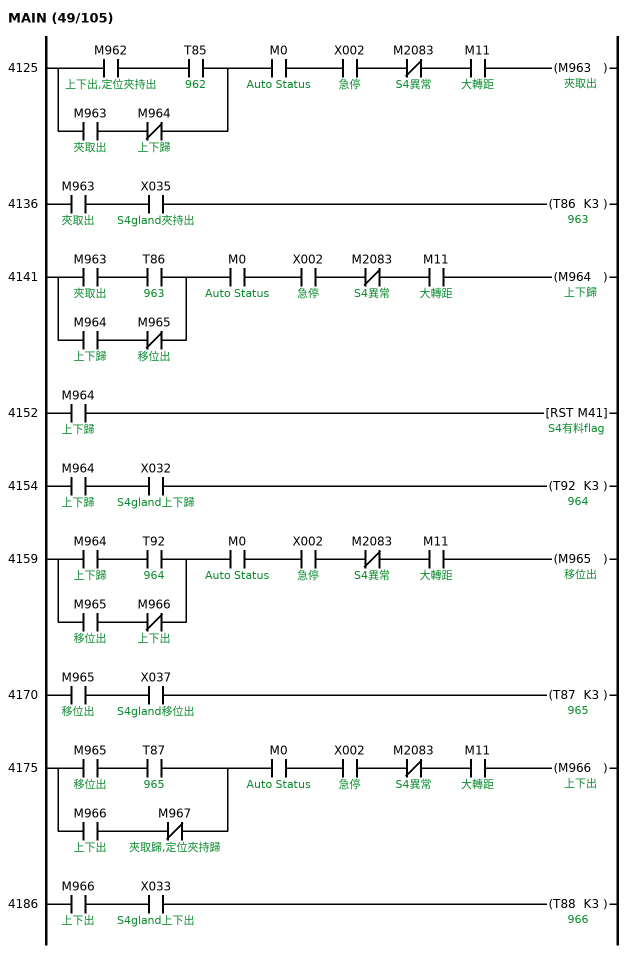
[picture p48: ladder of MAIN, rungs at steps 4125 to 4186]
4125  LD      M962  ; 上下出,定位夾持出
      AND     T85  ; 962
      LD      M963  ; 夾取出
      ANI     M964  ; 上下歸
      ORB
      AND     M0  ; Auto Status
      AND     X002  ; 急停
      ANI     M2083  ; S4異常
      AND     M11  ; 大轉距
      OUT     M963  ; 夾取出
4136  LD      M963  ; 夾取出
      AND     X035  ; S4gland夾持出
      OUT     T86 K3  ; 963
4141  LD      M963  ; 夾取出
      AND     T86  ; 963
      LD      M964  ; 上下歸
      ANI     M965  ; 移位出
      ORB
      AND     M0  ; Auto Status
      AND     X002  ; 急停
      ANI     M2083  ; S4異常
      AND     M11  ; 大轉距
      OUT     M964  ; 上下歸
4152  LD      M964  ; 上下歸
      RST     M41  ; S4有料flag
4154  LD      M964  ; 上下歸
      AND     X032  ; S4gland上下歸
      OUT     T92 K3  ; 964
4159  LD      M964  ; 上下歸
      AND     T92  ; 964
      LD      M965  ; 移位出
      ANI     M966  ; 上下出
      ORB
      AND     M0  ; Auto Status
      AND     X002  ; 急停
      ANI     M2083  ; S4異常
      AND     M11  ; 大轉距
      OUT     M965  ; 移位出
4170  LD      M965  ; 移位出
      AND     X037  ; S4gland移位出
      OUT     T87 K3  ; 965
4175  LD      M965  ; 移位出
      AND     T87  ; 965
      LD      M966  ; 上下出
      ANI     M967  ; 夾取歸,定位夾持歸
      ORB
      AND     M0  ; Auto Status
      AND     X002  ; 急停
      ANI     M2083  ; S4異常
      AND     M11  ; 大轉距
      OUT     M966  ; 上下出
4186  LD      M966  ; 上下出
      AND     X033  ; S4gland上下出
      OUT     T88 K3  ; 966
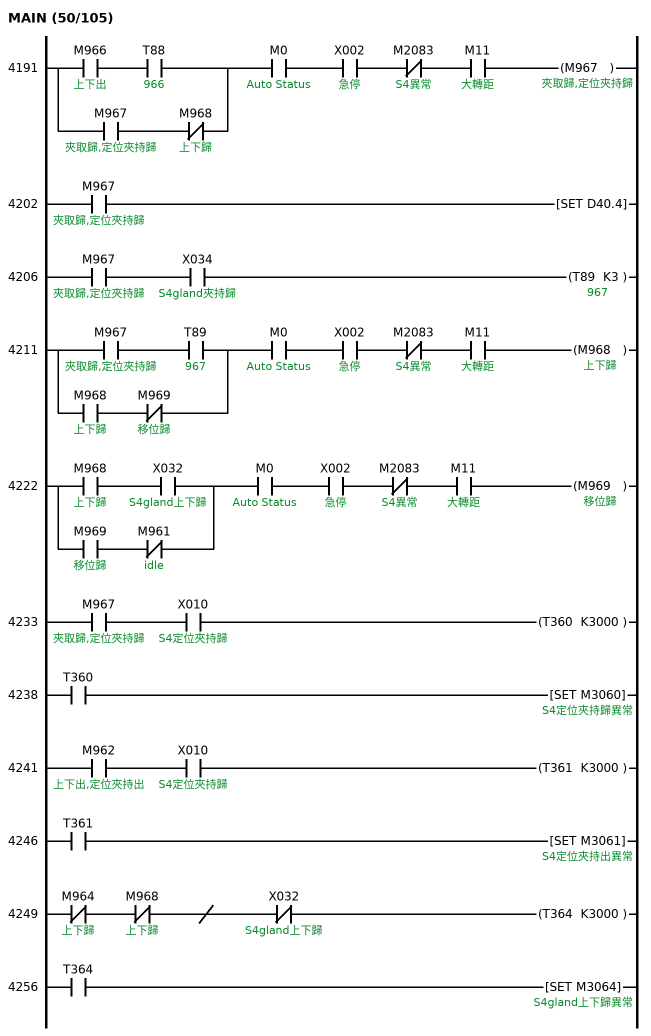
4191  LD      M966  ; 上下出
      AND     T88  ; 966
      LD      M967  ; 夾取歸,定位夾持歸
      ANI     M968  ; 上下歸
      ORB
      AND     M0  ; Auto Status
      AND     X002  ; 急停
      ANI     M2083  ; S4異常
      AND     M11  ; 大轉距
      OUT     M967  ; 夾取歸,定位夾持歸
4202  LD      M967  ; 夾取歸,定位夾持歸
      SET     D40.4
4206  LD      M967  ; 夾取歸,定位夾持歸
      AND     X034  ; S4gland夾持歸
      OUT     T89 K3  ; 967
4211  LD      M967  ; 夾取歸,定位夾持歸
      AND     T89  ; 967
      LD      M968  ; 上下歸
      ANI     M969  ; 移位歸
      ORB
      AND     M0  ; Auto Status
      AND     X002  ; 急停
      ANI     M2083  ; S4異常
      AND     M11  ; 大轉距
      OUT     M968  ; 上下歸
4222  LD      M968  ; 上下歸
      AND     X032  ; S4gland上下歸
      LD      M969  ; 移位歸
      ANI     M961  ; idle
      ORB
      AND     M0  ; Auto Status
      AND     X002  ; 急停
      ANI     M2083  ; S4異常
      AND     M11  ; 大轉距
      OUT     M969  ; 移位歸
4233  LD      M967  ; 夾取歸,定位夾持歸
      AND     X010  ; S4定位夾持歸
      OUT     T360 K3000
4238  LD      T360
      SET     M3060  ; S4定位夾持歸異常
4241  LD      M962  ; 上下出,定位夾持出
      AND     X010  ; S4定位夾持歸
      OUT     T361 K3000
4246  LD      T361
      SET     M3061  ; S4定位夾持出異常
4249  LDI     M964  ; 上下歸
      ANI     M968  ; 上下歸
      INV
      ANI     X032  ; S4gland上下歸
      OUT     T364 K3000
4256  LD      T364
      SET     M3064  ; S4gland上下歸異常
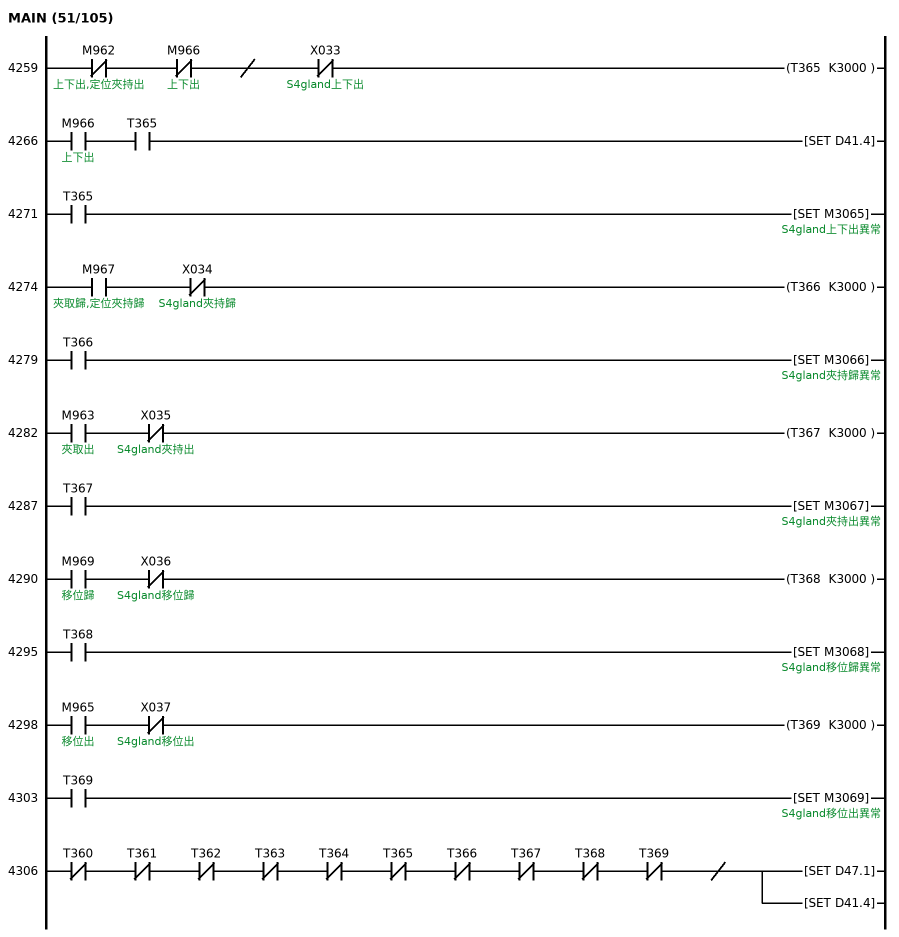
4259  LDI     M962  ; 上下出,定位夾持出
      ANI     M966  ; 上下出
      INV
      ANI     X033  ; S4gland上下出
      OUT     T365 K3000
4266  LD      M966  ; 上下出
      AND     T365
      SET     D41.4
4271  LD      T365
      SET     M3065  ; S4gland上下出異常
4274  LD      M967  ; 夾取歸,定位夾持歸
      ANI     X034  ; S4gland夾持歸
      OUT     T366 K3000
4279  LD      T366
      SET     M3066  ; S4gland夾持歸異常
4282  LD      M963  ; 夾取出
      ANI     X035  ; S4gland夾持出
      OUT     T367 K3000
4287  LD      T367
      SET     M3067  ; S4gland夾持出異常
4290  LD      M969  ; 移位歸
      ANI     X036  ; S4gland移位歸
      OUT     T368 K3000
4295  LD      T368
      SET     M3068  ; S4gland移位歸異常
4298  LD      M965  ; 移位出
      ANI     X037  ; S4gland移位出
      OUT     T369 K3000
4303  LD      T369
      SET     M3069  ; S4gland移位出異常
4306  LDI     T360
      ANI     T361
      ANI     T362
      ANI     T363
      ANI     T364
      ANI     T365
      ANI     T366
      ANI     T367
      ANI     T368
      ANI     T369
      INV
      SET     D47.1
      SET     D41.4
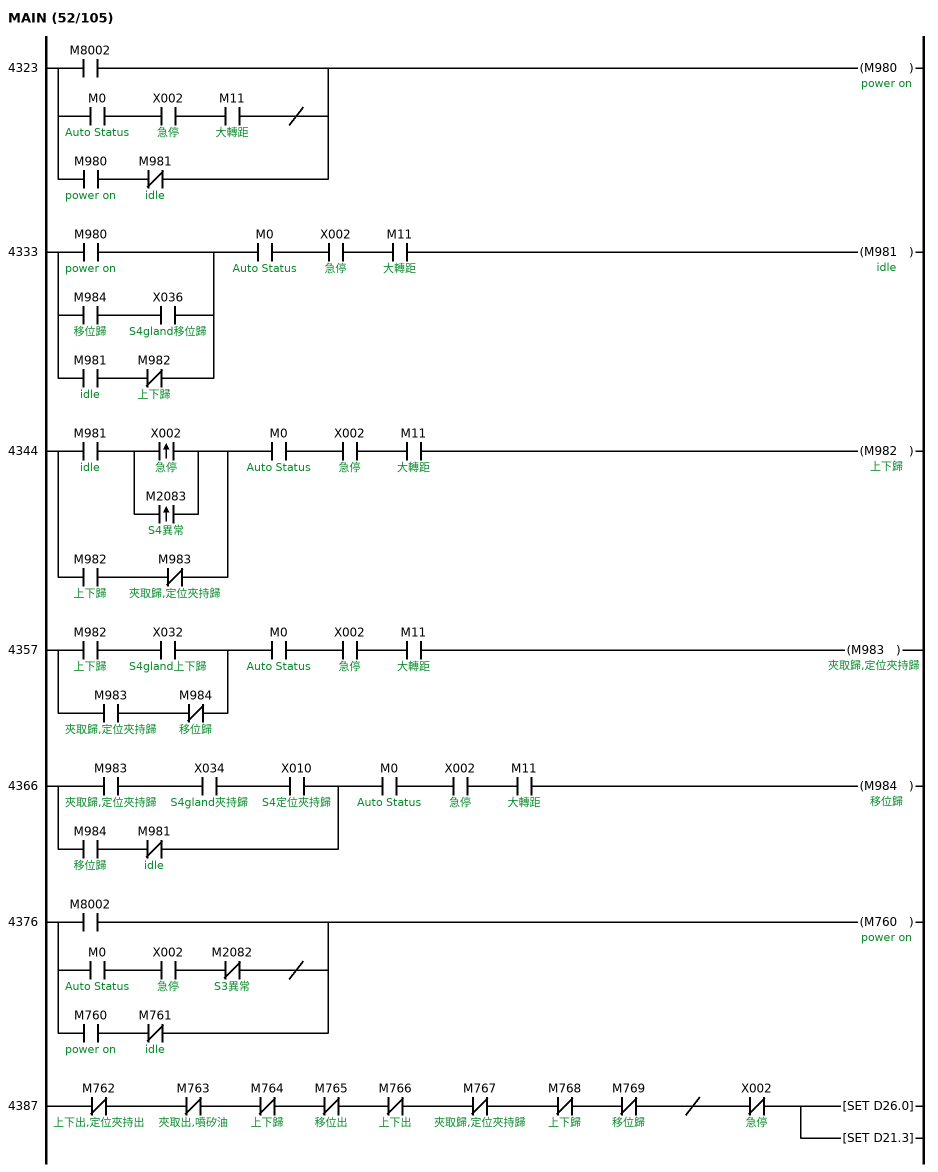
4323  LD      M8002
      LD      M0  ; Auto Status
      AND     X002  ; 急停
      AND     M11  ; 大轉距
      INV
      ORB
      LD      M980  ; power on
      ANI     M981  ; idle
      ORB
      OUT     M980  ; power on
4333  LD      M980  ; power on
      LD      M984  ; 移位歸
      AND     X036  ; S4gland移位歸
      ORB
      LD      M981  ; idle
      ANI     M982  ; 上下歸
      ORB
      AND     M0  ; Auto Status
      AND     X002  ; 急停
      AND     M11  ; 大轉距
      OUT     M981  ; idle
4344  LD      M981  ; idle
      LDP     X002  ; 急停
      ORP     M2083  ; S4異常
      ANB
      LD      M982  ; 上下歸
      ANI     M983  ; 夾取歸,定位夾持歸
      ORB
      AND     M0  ; Auto Status
      AND     X002  ; 急停
      AND     M11  ; 大轉距
      OUT     M982  ; 上下歸
4357  LD      M982  ; 上下歸
      AND     X032  ; S4gland上下歸
      LD      M983  ; 夾取歸,定位夾持歸
      ANI     M984  ; 移位歸
      ORB
      AND     M0  ; Auto Status
      AND     X002  ; 急停
      AND     M11  ; 大轉距
      OUT     M983  ; 夾取歸,定位夾持歸
4366  LD      M983  ; 夾取歸,定位夾持歸
      AND     X034  ; S4gland夾持歸
      AND     X010  ; S4定位夾持歸
      LD      M984  ; 移位歸
      ANI     M981  ; idle
      ORB
      AND     M0  ; Auto Status
      AND     X002  ; 急停
      AND     M11  ; 大轉距
      OUT     M984  ; 移位歸
4376  LD      M8002
      LD      M0  ; Auto Status
      AND     X002  ; 急停
      ANI     M2082  ; S3異常
      INV
      ORB
      LD      M760  ; power on
      ANI     M761  ; idle
      ORB
      OUT     M760  ; power on
4387  LDI     M762  ; 上下出,定位夾持出
      ANI     M763  ; 夾取出,噴矽油
      ANI     M764  ; 上下歸
      ANI     M765  ; 移位出
      ANI     M766  ; 上下出
      ANI     M767  ; 夾取歸,定位夾持歸
      ANI     M768  ; 上下歸
      ANI     M769  ; 移位歸
      INV
      ANI     X002  ; 急停
      SET     D26.0
      SET     D21.3
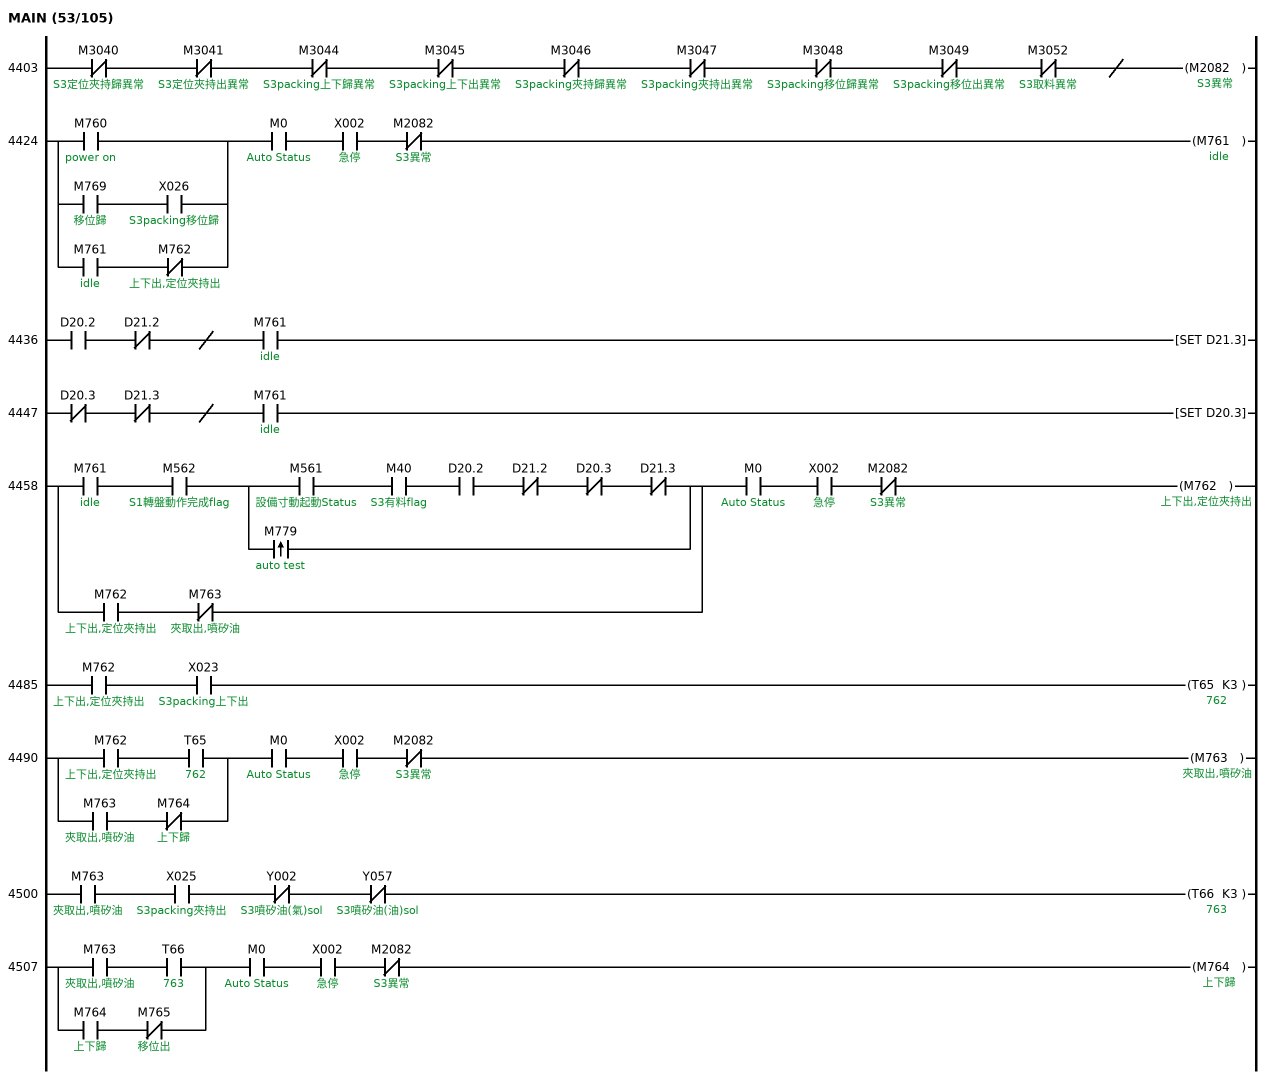
4403  LDI     M3040  ; S3定位夾持歸異常
      ANI     M3041  ; S3定位夾持出異常
      ANI     M3044  ; S3packing上下歸異常
      ANI     M3045  ; S3packing上下出異常
      ANI     M3046  ; S3packing夾持歸異常
      ANI     M3047  ; S3packing夾持出異常
      ANI     M3048  ; S3packing移位歸異常
      ANI     M3049  ; S3packing移位出異常
      ANI     M3052  ; S3取料異常
      INV
      OUT     M2082  ; S3異常
4424  LD      M760  ; power on
      LD      M769  ; 移位歸
      AND     X026  ; S3packing移位歸
      ORB
      LD      M761  ; idle
      ANI     M762  ; 上下出,定位夾持出
      ORB
      AND     M0  ; Auto Status
      AND     X002  ; 急停
      ANI     M2082  ; S3異常
      OUT     M761  ; idle
4436  LD      D20.2
      ANI     D21.2
      INV
      AND     M761  ; idle
      SET     D21.3
4447  LDI     D20.3
      ANI     D21.3
      INV
      AND     M761  ; idle
      SET     D20.3
4458  LD      M761  ; idle
      AND     M562  ; S1轉盤動作完成flag
      LD      M561  ; 設備寸動起動Status
      AND     M40  ; S3有料flag
      AND     D20.2
      ANI     D21.2
      ANI     D20.3
      ANI     D21.3
      ORP     M779  ; auto test
      ANB
      LD      M762  ; 上下出,定位夾持出
      ANI     M763  ; 夾取出,噴矽油
      ORB
      AND     M0  ; Auto Status
      AND     X002  ; 急停
      ANI     M2082  ; S3異常
      OUT     M762  ; 上下出,定位夾持出
4485  LD      M762  ; 上下出,定位夾持出
      AND     X023  ; S3packing上下出
      OUT     T65 K3  ; 762
4490  LD      M762  ; 上下出,定位夾持出
      AND     T65  ; 762
      LD      M763  ; 夾取出,噴矽油
      ANI     M764  ; 上下歸
      ORB
      AND     M0  ; Auto Status
      AND     X002  ; 急停
      ANI     M2082  ; S3異常
      OUT     M763  ; 夾取出,噴矽油
4500  LD      M763  ; 夾取出,噴矽油
      AND     X025  ; S3packing夾持出
      ANI     Y002  ; S3噴矽油(氣)sol
      ANI     Y057  ; S3噴矽油(油)sol
      OUT     T66 K3  ; 763
4507  LD      M763  ; 夾取出,噴矽油
      AND     T66  ; 763
      LD      M764  ; 上下歸
      ANI     M765  ; 移位出
      ORB
      AND     M0  ; Auto Status
      AND     X002  ; 急停
      ANI     M2082  ; S3異常
      OUT     M764  ; 上下歸
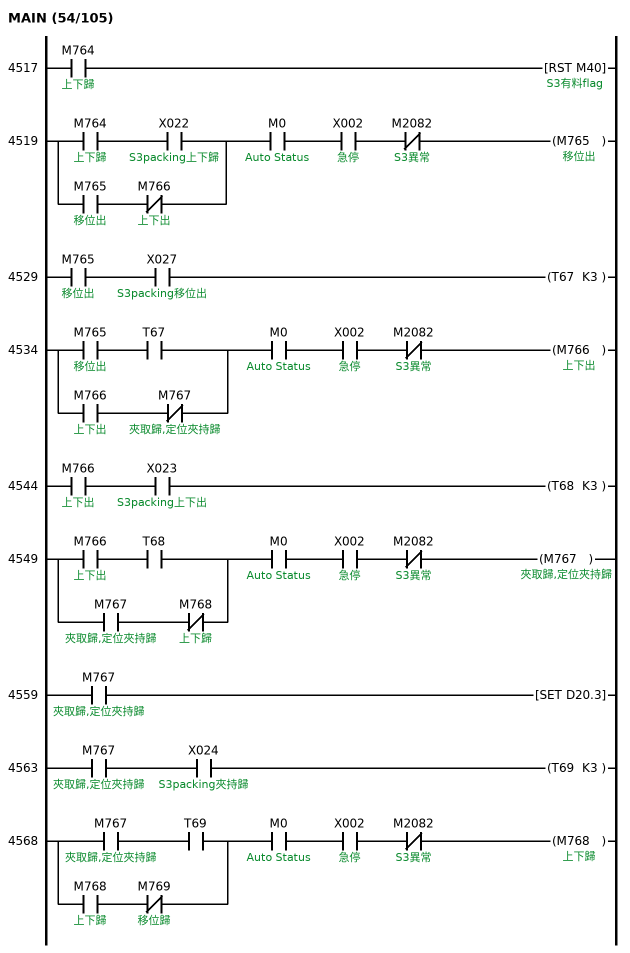
4517  LD      M764  ; 上下歸
      RST     M40  ; S3有料flag
4519  LD      M764  ; 上下歸
      AND     X022  ; S3packing上下歸
      LD      M765  ; 移位出
      ANI     M766  ; 上下出
      ORB
      AND     M0  ; Auto Status
      AND     X002  ; 急停
      ANI     M2082  ; S3異常
      OUT     M765  ; 移位出
4529  LD      M765  ; 移位出
      AND     X027  ; S3packing移位出
      OUT     T67 K3
4534  LD      M765  ; 移位出
      AND     T67
      LD      M766  ; 上下出
      ANI     M767  ; 夾取歸,定位夾持歸
      ORB
      AND     M0  ; Auto Status
      AND     X002  ; 急停
      ANI     M2082  ; S3異常
      OUT     M766  ; 上下出
4544  LD      M766  ; 上下出
      AND     X023  ; S3packing上下出
      OUT     T68 K3
4549  LD      M766  ; 上下出
      AND     T68
      LD      M767  ; 夾取歸,定位夾持歸
      ANI     M768  ; 上下歸
      ORB
      AND     M0  ; Auto Status
      AND     X002  ; 急停
      ANI     M2082  ; S3異常
      OUT     M767  ; 夾取歸,定位夾持歸
4559  LD      M767  ; 夾取歸,定位夾持歸
      SET     D20.3
4563  LD      M767  ; 夾取歸,定位夾持歸
      AND     X024  ; S3packing夾持歸
      OUT     T69 K3
4568  LD      M767  ; 夾取歸,定位夾持歸
      AND     T69
      LD      M768  ; 上下歸
      ANI     M769  ; 移位歸
      ORB
      AND     M0  ; Auto Status
      AND     X002  ; 急停
      ANI     M2082  ; S3異常
      OUT     M768  ; 上下歸
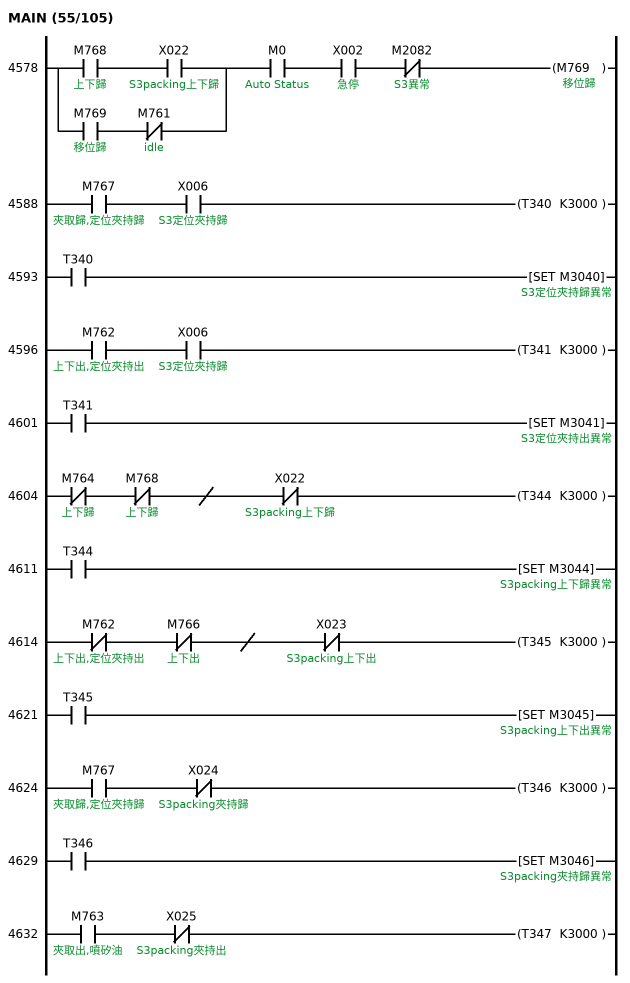
4578  LD      M768  ; 上下歸
      AND     X022  ; S3packing上下歸
      LD      M769  ; 移位歸
      ANI     M761  ; idle
      ORB
      AND     M0  ; Auto Status
      AND     X002  ; 急停
      ANI     M2082  ; S3異常
      OUT     M769  ; 移位歸
4588  LD      M767  ; 夾取歸,定位夾持歸
      AND     X006  ; S3定位夾持歸
      OUT     T340 K3000
4593  LD      T340
      SET     M3040  ; S3定位夾持歸異常
4596  LD      M762  ; 上下出,定位夾持出
      AND     X006  ; S3定位夾持歸
      OUT     T341 K3000
4601  LD      T341
      SET     M3041  ; S3定位夾持出異常
4604  LDI     M764  ; 上下歸
      ANI     M768  ; 上下歸
      INV
      ANI     X022  ; S3packing上下歸
      OUT     T344 K3000
4611  LD      T344
      SET     M3044  ; S3packing上下歸異常
4614  LDI     M762  ; 上下出,定位夾持出
      ANI     M766  ; 上下出
      INV
      ANI     X023  ; S3packing上下出
      OUT     T345 K3000
4621  LD      T345
      SET     M3045  ; S3packing上下出異常
4624  LD      M767  ; 夾取歸,定位夾持歸
      ANI     X024  ; S3packing夾持歸
      OUT     T346 K3000
4629  LD      T346
      SET     M3046  ; S3packing夾持歸異常
4632  LD      M763  ; 夾取出,噴矽油
      ANI     X025  ; S3packing夾持出
      OUT     T347 K3000
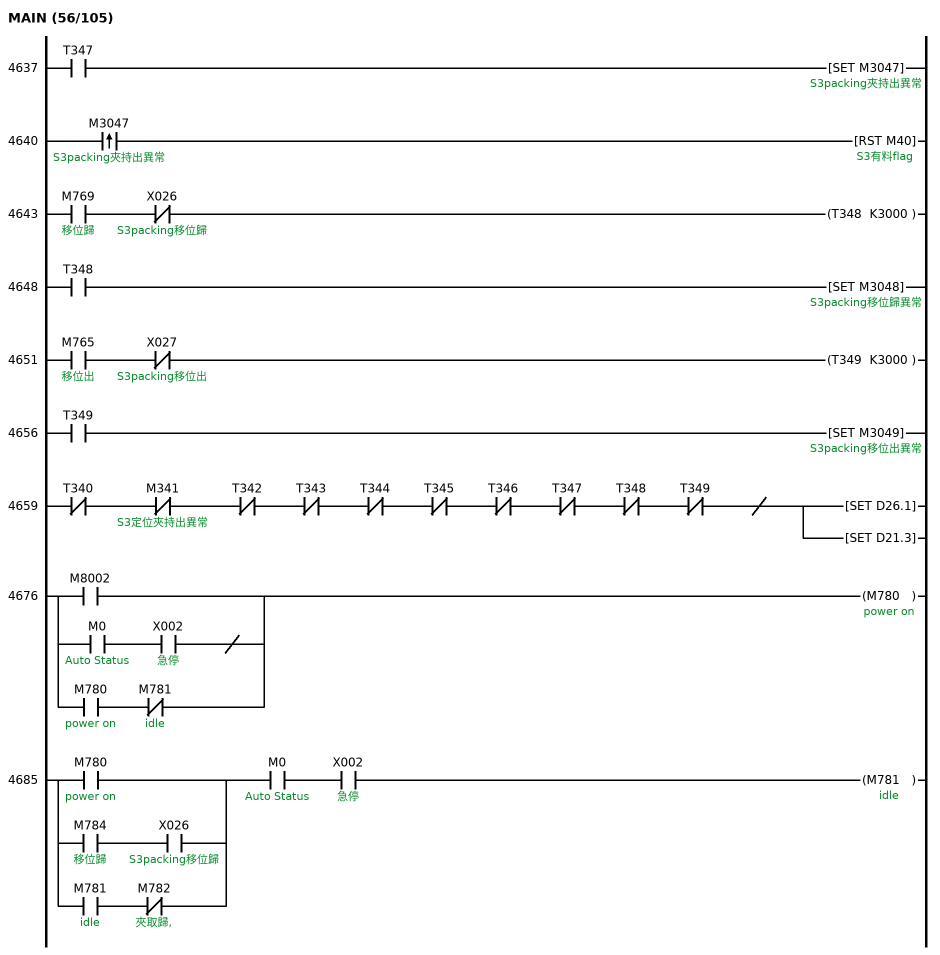
4637  LD      T347
      SET     M3047  ; S3packing夾持出異常
4640  LDP     M3047  ; S3packing夾持出異常
      RST     M40  ; S3有料flag
4643  LD      M769  ; 移位歸
      ANI     X026  ; S3packing移位歸
      OUT     T348 K3000
4648  LD      T348
      SET     M3048  ; S3packing移位歸異常
4651  LD      M765  ; 移位出
      ANI     X027  ; S3packing移位出
      OUT     T349 K3000
4656  LD      T349
      SET     M3049  ; S3packing移位出異常
4659  LDI     T340
      ANI     M341  ; S3定位夾持出異常
      ANI     T342
      ANI     T343
      ANI     T344
      ANI     T345
      ANI     T346
      ANI     T347
      ANI     T348
      ANI     T349
      INV
      SET     D26.1
      SET     D21.3
4676  LD      M8002
      LD      M0  ; Auto Status
      AND     X002  ; 急停
      INV
      ORB
      LD      M780  ; power on
      ANI     M781  ; idle
      ORB
      OUT     M780  ; power on
4685  LD      M780  ; power on
      LD      M784  ; 移位歸
      AND     X026  ; S3packing移位歸
      ORB
      LD      M781  ; idle
      ANI     M782  ; 夾取歸,
      ORB
      AND     M0  ; Auto Status
      AND     X002  ; 急停
      OUT     M781  ; idle
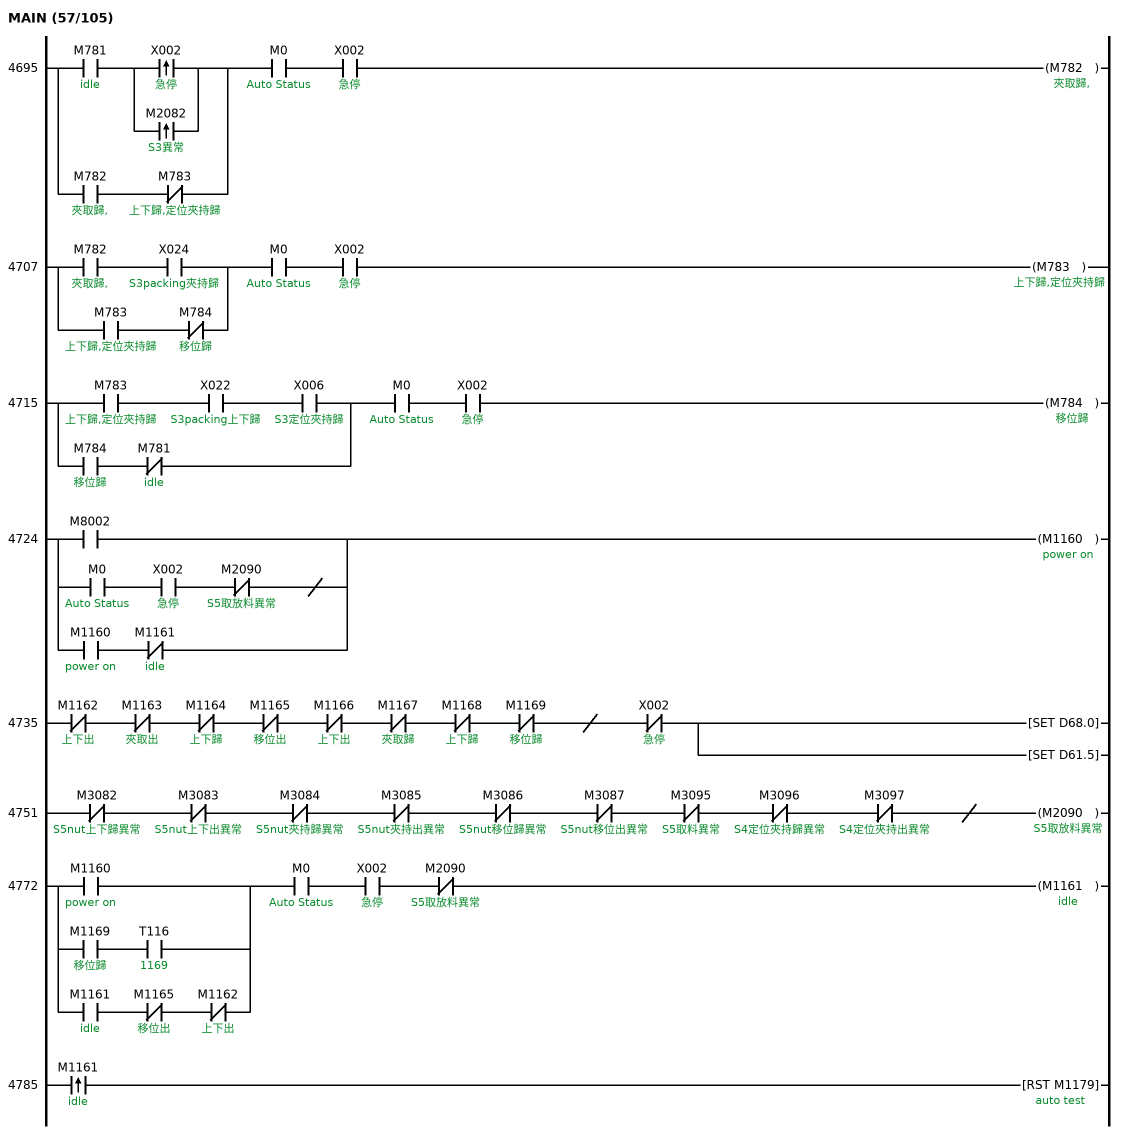
4695  LD      M781  ; idle
      LDP     X002  ; 急停
      ORP     M2082  ; S3異常
      ANB
      LD      M782  ; 夾取歸,
      ANI     M783  ; 上下歸,定位夾持歸
      ORB
      AND     M0  ; Auto Status
      AND     X002  ; 急停
      OUT     M782  ; 夾取歸,
4707  LD      M782  ; 夾取歸,
      AND     X024  ; S3packing夾持歸
      LD      M783  ; 上下歸,定位夾持歸
      ANI     M784  ; 移位歸
      ORB
      AND     M0  ; Auto Status
      AND     X002  ; 急停
      OUT     M783  ; 上下歸,定位夾持歸
4715  LD      M783  ; 上下歸,定位夾持歸
      AND     X022  ; S3packing上下歸
      AND     X006  ; S3定位夾持歸
      LD      M784  ; 移位歸
      ANI     M781  ; idle
      ORB
      AND     M0  ; Auto Status
      AND     X002  ; 急停
      OUT     M784  ; 移位歸
4724  LD      M8002
      LD      M0  ; Auto Status
      AND     X002  ; 急停
      ANI     M2090  ; S5取放料異常
      INV
      ORB
      LD      M1160  ; power on
      ANI     M1161  ; idle
      ORB
      OUT     M1160  ; power on
4735  LDI     M1162  ; 上下出
      ANI     M1163  ; 夾取出
      ANI     M1164  ; 上下歸
      ANI     M1165  ; 移位出
      ANI     M1166  ; 上下出
      ANI     M1167  ; 夾取歸
      ANI     M1168  ; 上下歸
      ANI     M1169  ; 移位歸
      INV
      ANI     X002  ; 急停
      SET     D68.0
      SET     D61.5
4751  LDI     M3082  ; S5nut上下歸異常
      ANI     M3083  ; S5nut上下出異常
      ANI     M3084  ; S5nut夾持歸異常
      ANI     M3085  ; S5nut夾持出異常
      ANI     M3086  ; S5nut移位歸異常
      ANI     M3087  ; S5nut移位出異常
      ANI     M3095  ; S5取料異常
      ANI     M3096  ; S4定位夾持歸異常
      ANI     M3097  ; S4定位夾持出異常
      INV
      OUT     M2090  ; S5取放料異常
4772  LD      M1160  ; power on
      LD      M1169  ; 移位歸
      AND     T116  ; 1169
      ORB
      LD      M1161  ; idle
      ANI     M1165  ; 移位出
      ANI     M1162  ; 上下出
      ORB
      AND     M0  ; Auto Status
      AND     X002  ; 急停
      ANI     M2090  ; S5取放料異常
      OUT     M1161  ; idle
4785  LDP     M1161  ; idle
      RST     M1179  ; auto test
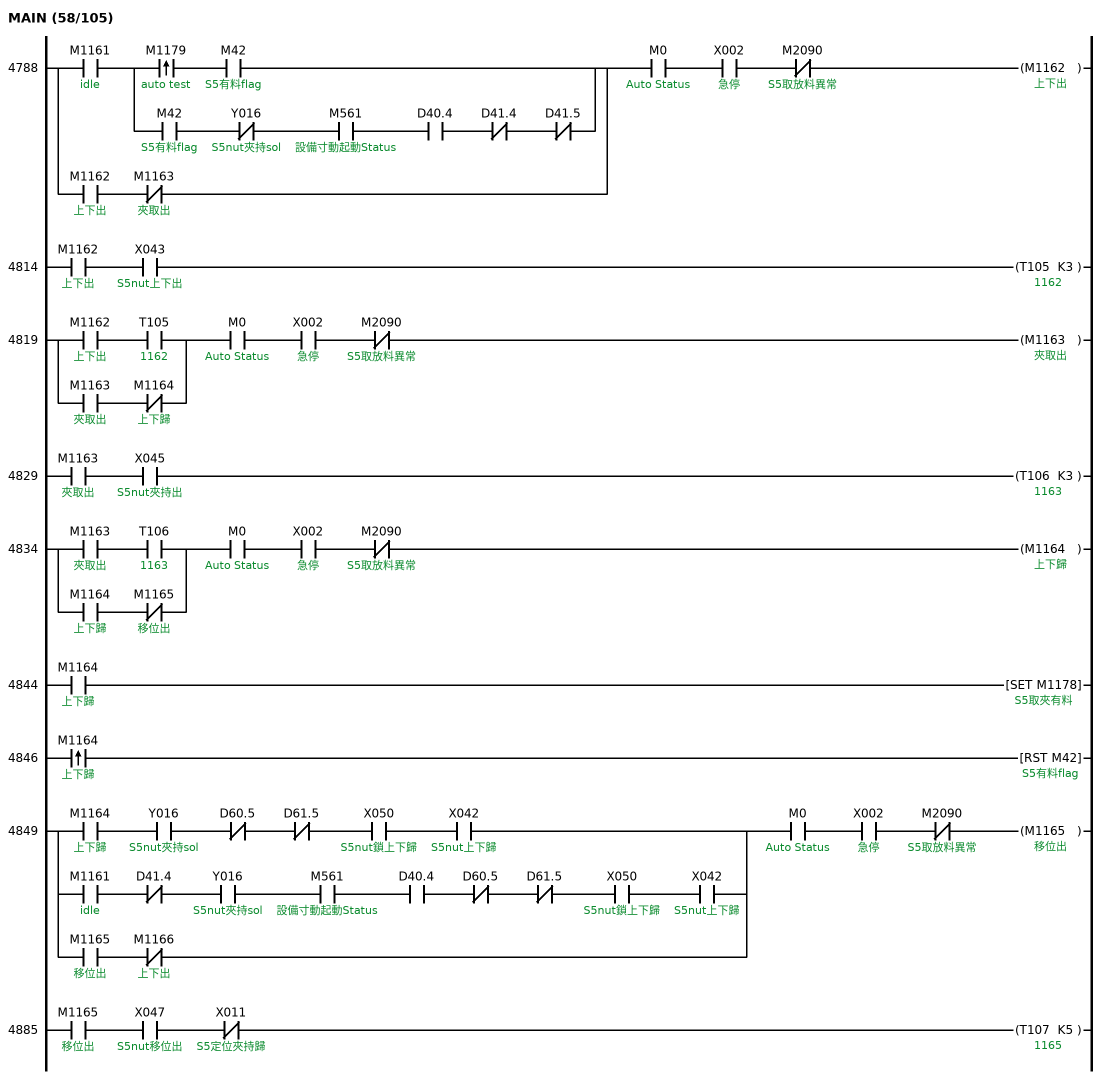
4788  LD      M1161  ; idle
      LDP     M1179  ; auto test
      AND     M42  ; S5有料flag
      LD      M42  ; S5有料flag
      ANI     Y016  ; S5nut夾持sol
      AND     M561  ; 設備寸動起動Status
      AND     D40.4
      ANI     D41.4
      ANI     D41.5
      ORB
      ANB
      LD      M1162  ; 上下出
      ANI     M1163  ; 夾取出
      ORB
      AND     M0  ; Auto Status
      AND     X002  ; 急停
      ANI     M2090  ; S5取放料異常
      OUT     M1162  ; 上下出
4814  LD      M1162  ; 上下出
      AND     X043  ; S5nut上下出
      OUT     T105 K3  ; 1162
4819  LD      M1162  ; 上下出
      AND     T105  ; 1162
      LD      M1163  ; 夾取出
      ANI     M1164  ; 上下歸
      ORB
      AND     M0  ; Auto Status
      AND     X002  ; 急停
      ANI     M2090  ; S5取放料異常
      OUT     M1163  ; 夾取出
4829  LD      M1163  ; 夾取出
      AND     X045  ; S5nut夾持出
      OUT     T106 K3  ; 1163
4834  LD      M1163  ; 夾取出
      AND     T106  ; 1163
      LD      M1164  ; 上下歸
      ANI     M1165  ; 移位出
      ORB
      AND     M0  ; Auto Status
      AND     X002  ; 急停
      ANI     M2090  ; S5取放料異常
      OUT     M1164  ; 上下歸
4844  LD      M1164  ; 上下歸
      SET     M1178  ; S5取夾有料
4846  LDP     M1164  ; 上下歸
      RST     M42  ; S5有料flag
4849  LD      M1164  ; 上下歸
      AND     Y016  ; S5nut夾持sol
      ANI     D60.5
      ANI     D61.5
      AND     X050  ; S5nut鎖上下歸
      AND     X042  ; S5nut上下歸
      LD      M1161  ; idle
      ANI     D41.4
      AND     Y016  ; S5nut夾持sol
      AND     M561  ; 設備寸動起動Status
      AND     D40.4
      ANI     D60.5
      ANI     D61.5
      AND     X050  ; S5nut鎖上下歸
      AND     X042  ; S5nut上下歸
      ORB
      LD      M1165  ; 移位出
      ANI     M1166  ; 上下出
      ORB
      AND     M0  ; Auto Status
      AND     X002  ; 急停
      ANI     M2090  ; S5取放料異常
      OUT     M1165  ; 移位出
4885  LD      M1165  ; 移位出
      AND     X047  ; S5nut移位出
      ANI     X011  ; S5定位夾持歸
      OUT     T107 K5  ; 1165
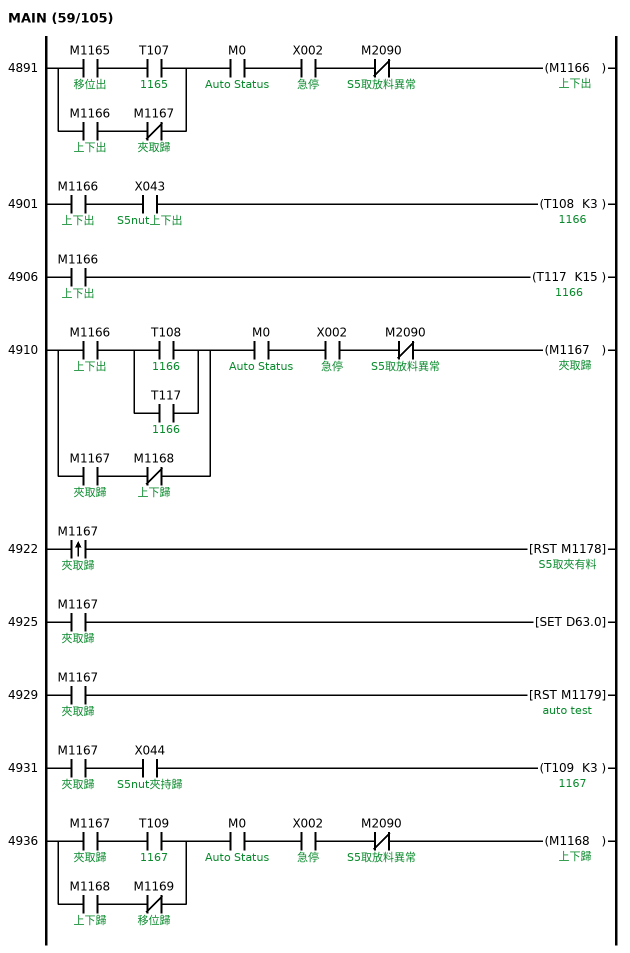
4891  LD      M1165  ; 移位出
      AND     T107  ; 1165
      LD      M1166  ; 上下出
      ANI     M1167  ; 夾取歸
      ORB
      AND     M0  ; Auto Status
      AND     X002  ; 急停
      ANI     M2090  ; S5取放料異常
      OUT     M1166  ; 上下出
4901  LD      M1166  ; 上下出
      AND     X043  ; S5nut上下出
      OUT     T108 K3  ; 1166
4906  LD      M1166  ; 上下出
      OUT     T117 K15  ; 1166
4910  LD      M1166  ; 上下出
      LD      T108  ; 1166
      OR      T117  ; 1166
      ANB
      LD      M1167  ; 夾取歸
      ANI     M1168  ; 上下歸
      ORB
      AND     M0  ; Auto Status
      AND     X002  ; 急停
      ANI     M2090  ; S5取放料異常
      OUT     M1167  ; 夾取歸
4922  LDP     M1167  ; 夾取歸
      RST     M1178  ; S5取夾有料
4925  LD      M1167  ; 夾取歸
      SET     D63.0
4929  LD      M1167  ; 夾取歸
      RST     M1179  ; auto test
4931  LD      M1167  ; 夾取歸
      AND     X044  ; S5nut夾持歸
      OUT     T109 K3  ; 1167
4936  LD      M1167  ; 夾取歸
      AND     T109  ; 1167
      LD      M1168  ; 上下歸
      ANI     M1169  ; 移位歸
      ORB
      AND     M0  ; Auto Status
      AND     X002  ; 急停
      ANI     M2090  ; S5取放料異常
      OUT     M1168  ; 上下歸
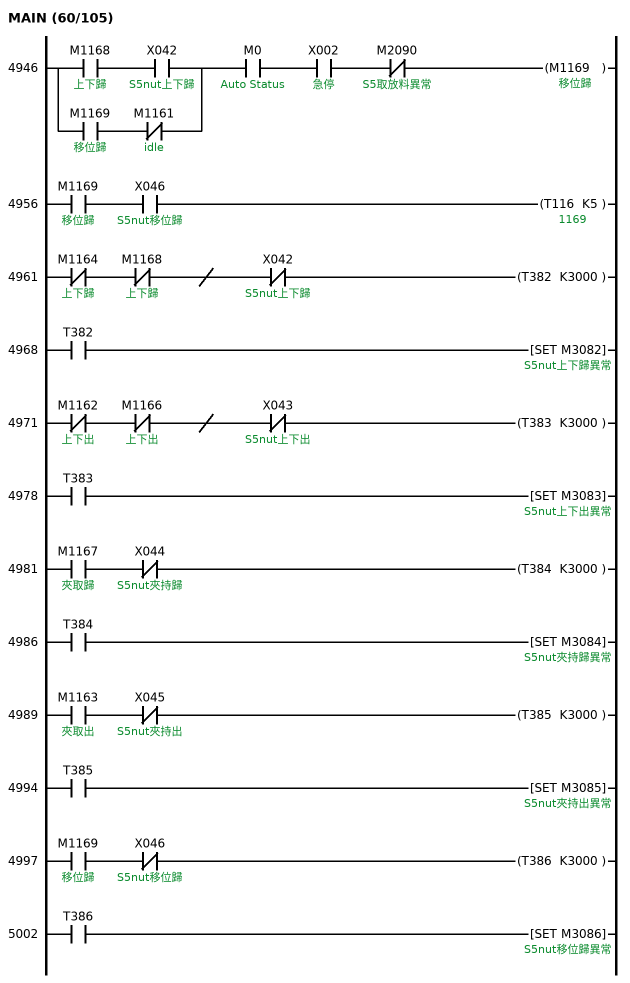
4946  LD      M1168  ; 上下歸
      AND     X042  ; S5nut上下歸
      LD      M1169  ; 移位歸
      ANI     M1161  ; idle
      ORB
      AND     M0  ; Auto Status
      AND     X002  ; 急停
      ANI     M2090  ; S5取放料異常
      OUT     M1169  ; 移位歸
4956  LD      M1169  ; 移位歸
      AND     X046  ; S5nut移位歸
      OUT     T116 K5  ; 1169
4961  LDI     M1164  ; 上下歸
      ANI     M1168  ; 上下歸
      INV
      ANI     X042  ; S5nut上下歸
      OUT     T382 K3000
4968  LD      T382
      SET     M3082  ; S5nut上下歸異常
4971  LDI     M1162  ; 上下出
      ANI     M1166  ; 上下出
      INV
      ANI     X043  ; S5nut上下出
      OUT     T383 K3000
4978  LD      T383
      SET     M3083  ; S5nut上下出異常
4981  LD      M1167  ; 夾取歸
      ANI     X044  ; S5nut夾持歸
      OUT     T384 K3000
4986  LD      T384
      SET     M3084  ; S5nut夾持歸異常
4989  LD      M1163  ; 夾取出
      ANI     X045  ; S5nut夾持出
      OUT     T385 K3000
4994  LD      T385
      SET     M3085  ; S5nut夾持出異常
4997  LD      M1169  ; 移位歸
      ANI     X046  ; S5nut移位歸
      OUT     T386 K3000
5002  LD      T386
      SET     M3086  ; S5nut移位歸異常
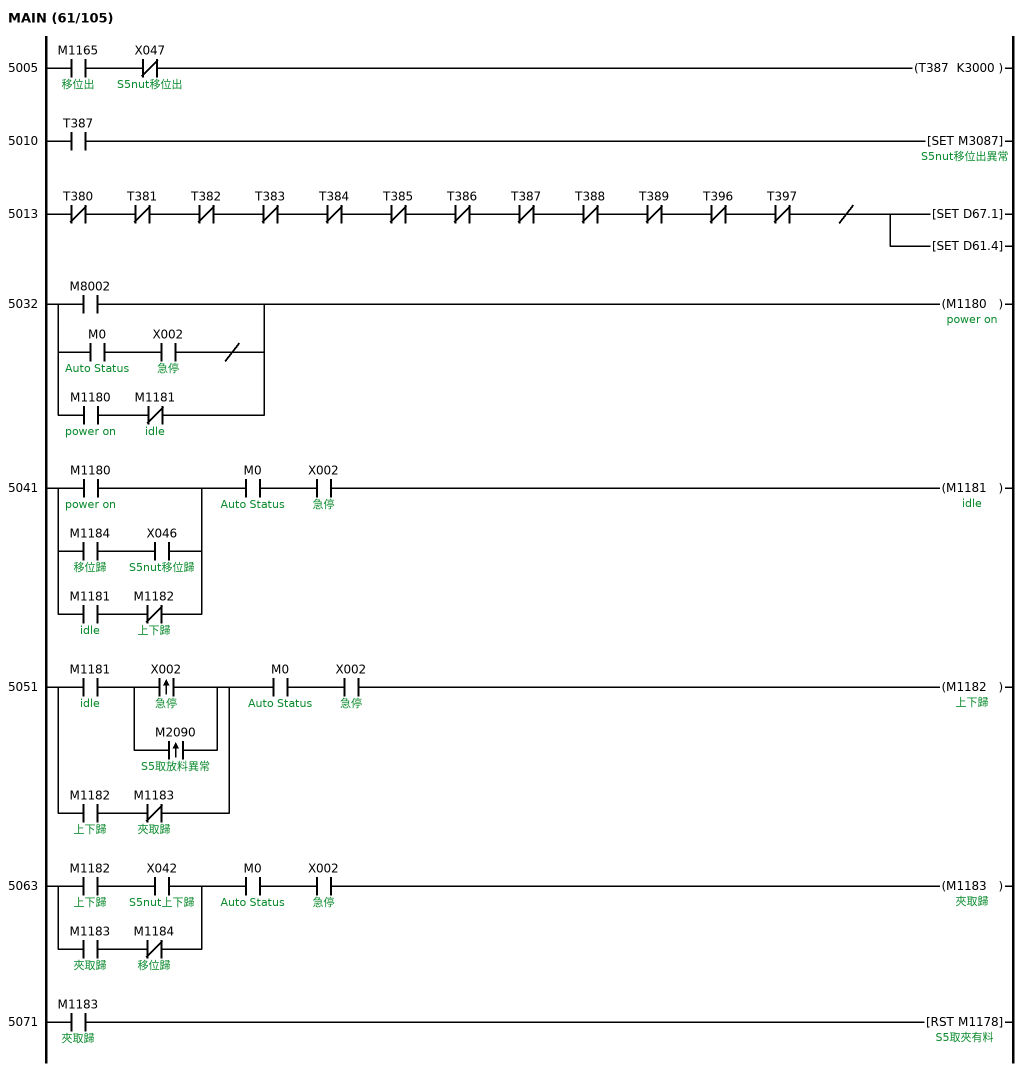
5005  LD      M1165  ; 移位出
      ANI     X047  ; S5nut移位出
      OUT     T387 K3000
5010  LD      T387
      SET     M3087  ; S5nut移位出異常
5013  LDI     T380
      ANI     T381
      ANI     T382
      ANI     T383
      ANI     T384
      ANI     T385
      ANI     T386
      ANI     T387
      ANI     T388
      ANI     T389
      ANI     T396
      ANI     T397
      INV
      SET     D67.1
      SET     D61.4
5032  LD      M8002
      LD      M0  ; Auto Status
      AND     X002  ; 急停
      INV
      ORB
      LD      M1180  ; power on
      ANI     M1181  ; idle
      ORB
      OUT     M1180  ; power on
5041  LD      M1180  ; power on
      LD      M1184  ; 移位歸
      AND     X046  ; S5nut移位歸
      ORB
      LD      M1181  ; idle
      ANI     M1182  ; 上下歸
      ORB
      AND     M0  ; Auto Status
      AND     X002  ; 急停
      OUT     M1181  ; idle
5051  LD      M1181  ; idle
      LDP     X002  ; 急停
      ORP     M2090  ; S5取放料異常
      ANB
      LD      M1182  ; 上下歸
      ANI     M1183  ; 夾取歸
      ORB
      AND     M0  ; Auto Status
      AND     X002  ; 急停
      OUT     M1182  ; 上下歸
5063  LD      M1182  ; 上下歸
      AND     X042  ; S5nut上下歸
      LD      M1183  ; 夾取歸
      ANI     M1184  ; 移位歸
      ORB
      AND     M0  ; Auto Status
      AND     X002  ; 急停
      OUT     M1183  ; 夾取歸
5071  LD      M1183  ; 夾取歸
      RST     M1178  ; S5取夾有料
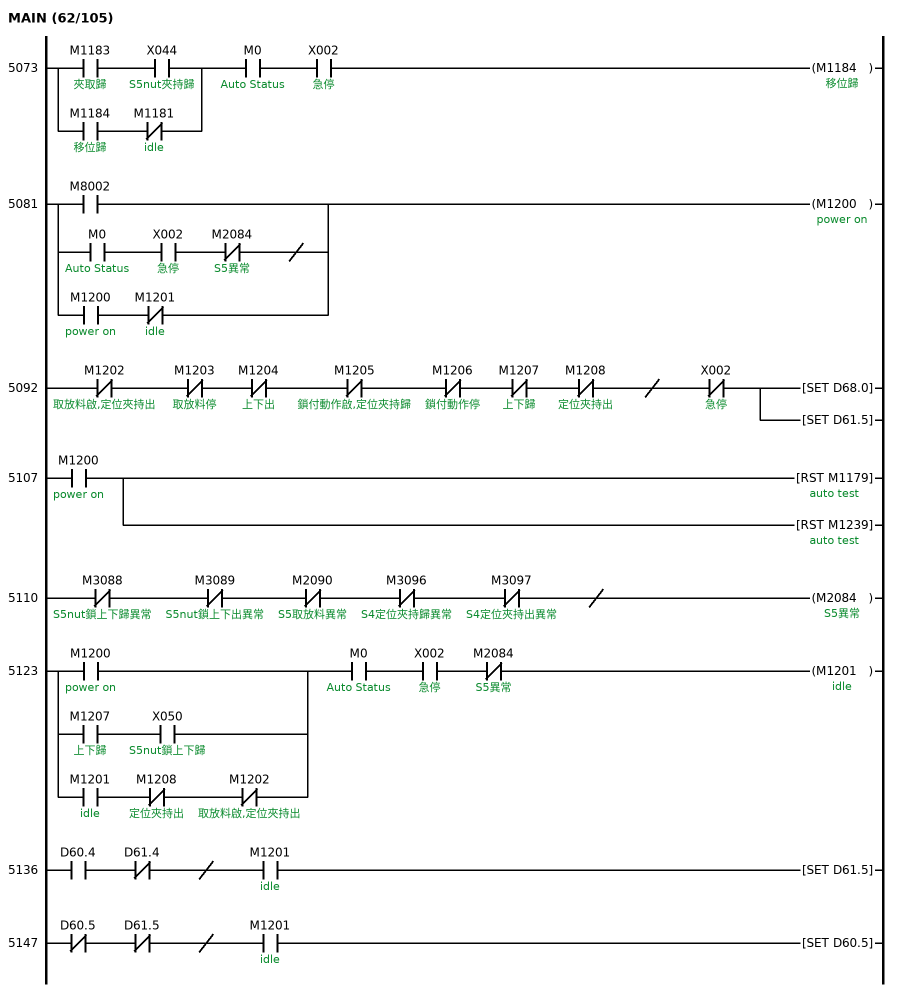
5073  LD      M1183  ; 夾取歸
      AND     X044  ; S5nut夾持歸
      LD      M1184  ; 移位歸
      ANI     M1181  ; idle
      ORB
      AND     M0  ; Auto Status
      AND     X002  ; 急停
      OUT     M1184  ; 移位歸
5081  LD      M8002
      LD      M0  ; Auto Status
      AND     X002  ; 急停
      ANI     M2084  ; S5異常
      INV
      ORB
      LD      M1200  ; power on
      ANI     M1201  ; idle
      ORB
      OUT     M1200  ; power on
5092  LDI     M1202  ; 取放料啟,定位夾持出
      ANI     M1203  ; 取放料停
      ANI     M1204  ; 上下出
      ANI     M1205  ; 鎖付動作啟,定位夾持歸
      ANI     M1206  ; 鎖付動作停
      ANI     M1207  ; 上下歸
      ANI     M1208  ; 定位夾持出
      INV
      ANI     X002  ; 急停
      SET     D68.0
      SET     D61.5
5107  LD      M1200  ; power on
      RST     M1179  ; auto test
      RST     M1239  ; auto test
5110  LDI     M3088  ; S5nut鎖上下歸異常
      ANI     M3089  ; S5nut鎖上下出異常
      ANI     M2090  ; S5取放料異常
      ANI     M3096  ; S4定位夾持歸異常
      ANI     M3097  ; S4定位夾持出異常
      INV
      OUT     M2084  ; S5異常
5123  LD      M1200  ; power on
      LD      M1207  ; 上下歸
      AND     X050  ; S5nut鎖上下歸
      ORB
      LD      M1201  ; idle
      ANI     M1208  ; 定位夾持出
      ANI     M1202  ; 取放料啟,定位夾持出
      ORB
      AND     M0  ; Auto Status
      AND     X002  ; 急停
      ANI     M2084  ; S5異常
      OUT     M1201  ; idle
5136  LD      D60.4
      ANI     D61.4
      INV
      AND     M1201  ; idle
      SET     D61.5
5147  LDI     D60.5
      ANI     D61.5
      INV
      AND     M1201  ; idle
      SET     D60.5
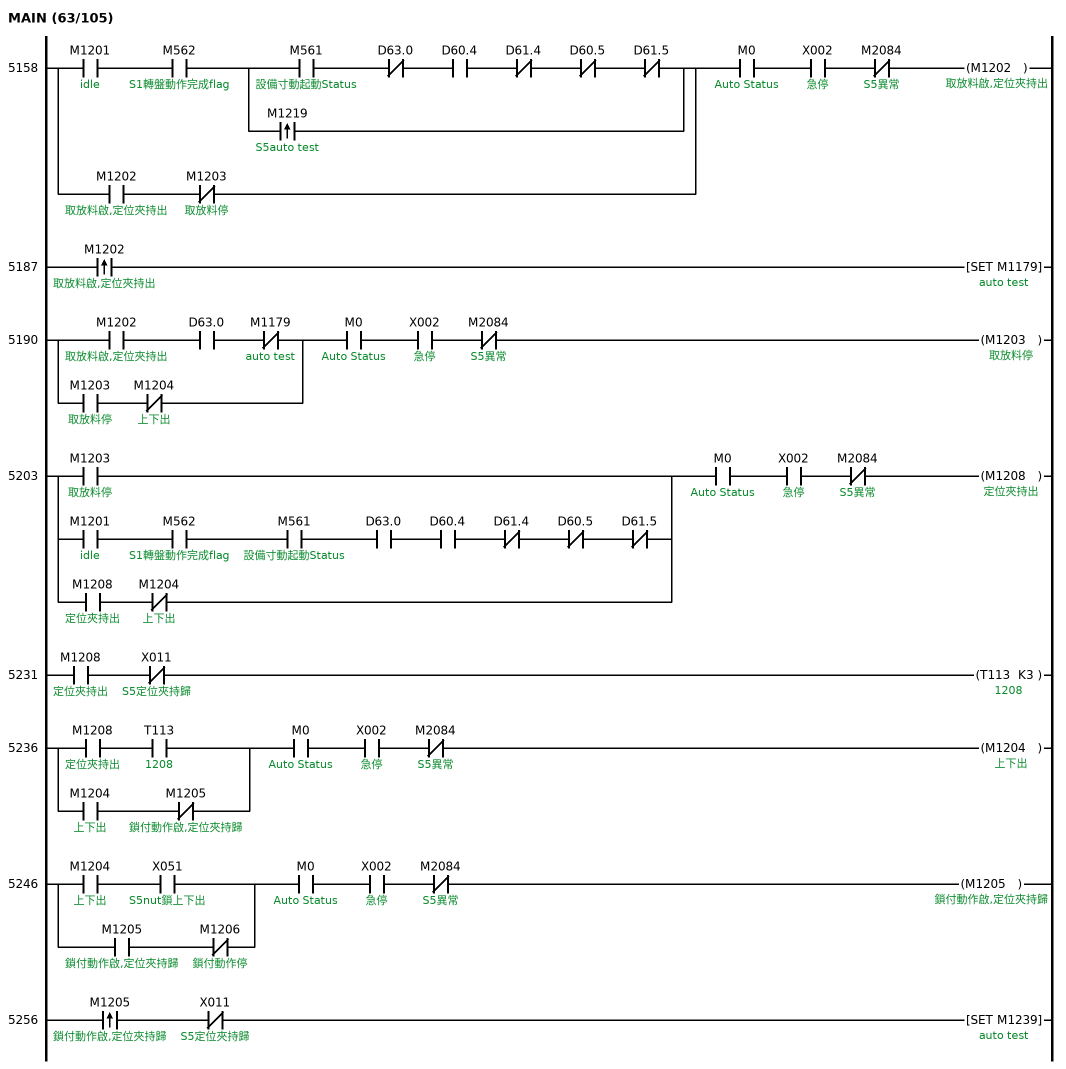
5158  LD      M1201  ; idle
      AND     M562  ; S1轉盤動作完成flag
      LD      M561  ; 設備寸動起動Status
      ANI     D63.0
      AND     D60.4
      ANI     D61.4
      ANI     D60.5
      ANI     D61.5
      ORP     M1219  ; S5auto test
      ANB
      LD      M1202  ; 取放料啟,定位夾持出
      ANI     M1203  ; 取放料停
      ORB
      AND     M0  ; Auto Status
      AND     X002  ; 急停
      ANI     M2084  ; S5異常
      OUT     M1202  ; 取放料啟,定位夾持出
5187  LDP     M1202  ; 取放料啟,定位夾持出
      SET     M1179  ; auto test
5190  LD      M1202  ; 取放料啟,定位夾持出
      AND     D63.0
      ANI     M1179  ; auto test
      LD      M1203  ; 取放料停
      ANI     M1204  ; 上下出
      ORB
      AND     M0  ; Auto Status
      AND     X002  ; 急停
      ANI     M2084  ; S5異常
      OUT     M1203  ; 取放料停
5203  LD      M1203  ; 取放料停
      LD      M1201  ; idle
      AND     M562  ; S1轉盤動作完成flag
      AND     M561  ; 設備寸動起動Status
      AND     D63.0
      AND     D60.4
      ANI     D61.4
      ANI     D60.5
      ANI     D61.5
      ORB
      LD      M1208  ; 定位夾持出
      ANI     M1204  ; 上下出
      ORB
      AND     M0  ; Auto Status
      AND     X002  ; 急停
      ANI     M2084  ; S5異常
      OUT     M1208  ; 定位夾持出
5231  LD      M1208  ; 定位夾持出
      ANI     X011  ; S5定位夾持歸
      OUT     T113 K3  ; 1208
5236  LD      M1208  ; 定位夾持出
      AND     T113  ; 1208
      LD      M1204  ; 上下出
      ANI     M1205  ; 鎖付動作啟,定位夾持歸
      ORB
      AND     M0  ; Auto Status
      AND     X002  ; 急停
      ANI     M2084  ; S5異常
      OUT     M1204  ; 上下出
5246  LD      M1204  ; 上下出
      AND     X051  ; S5nut鎖上下出
      LD      M1205  ; 鎖付動作啟,定位夾持歸
      ANI     M1206  ; 鎖付動作停
      ORB
      AND     M0  ; Auto Status
      AND     X002  ; 急停
      ANI     M2084  ; S5異常
      OUT     M1205  ; 鎖付動作啟,定位夾持歸
5256  LDP     M1205  ; 鎖付動作啟,定位夾持歸
      ANI     X011  ; S5定位夾持歸
      SET     M1239  ; auto test
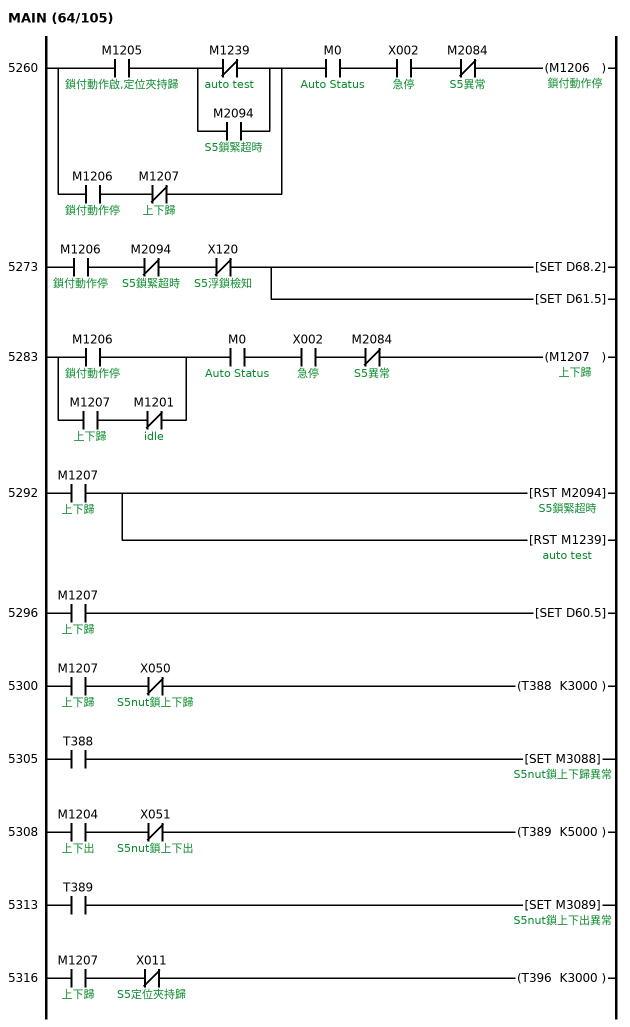
5260  LD      M1205  ; 鎖付動作啟,定位夾持歸
      LDI     M1239  ; auto test
      OR      M2094  ; S5鎖緊超時
      ANB
      LD      M1206  ; 鎖付動作停
      ANI     M1207  ; 上下歸
      ORB
      AND     M0  ; Auto Status
      AND     X002  ; 急停
      ANI     M2084  ; S5異常
      OUT     M1206  ; 鎖付動作停
5273  LD      M1206  ; 鎖付動作停
      ANI     M2094  ; S5鎖緊超時
      ANI     X120  ; S5浮鎖檢知
      SET     D68.2
      SET     D61.5
5283  LD      M1206  ; 鎖付動作停
      LD      M1207  ; 上下歸
      ANI     M1201  ; idle
      ORB
      AND     M0  ; Auto Status
      AND     X002  ; 急停
      ANI     M2084  ; S5異常
      OUT     M1207  ; 上下歸
5292  LD      M1207  ; 上下歸
      RST     M2094  ; S5鎖緊超時
      RST     M1239  ; auto test
5296  LD      M1207  ; 上下歸
      SET     D60.5
5300  LD      M1207  ; 上下歸
      ANI     X050  ; S5nut鎖上下歸
      OUT     T388 K3000
5305  LD      T388
      SET     M3088  ; S5nut鎖上下歸異常
5308  LD      M1204  ; 上下出
      ANI     X051  ; S5nut鎖上下出
      OUT     T389 K5000
5313  LD      T389
      SET     M3089  ; S5nut鎖上下出異常
5316  LD      M1207  ; 上下歸
      ANI     X011  ; S5定位夾持歸
      OUT     T396 K3000
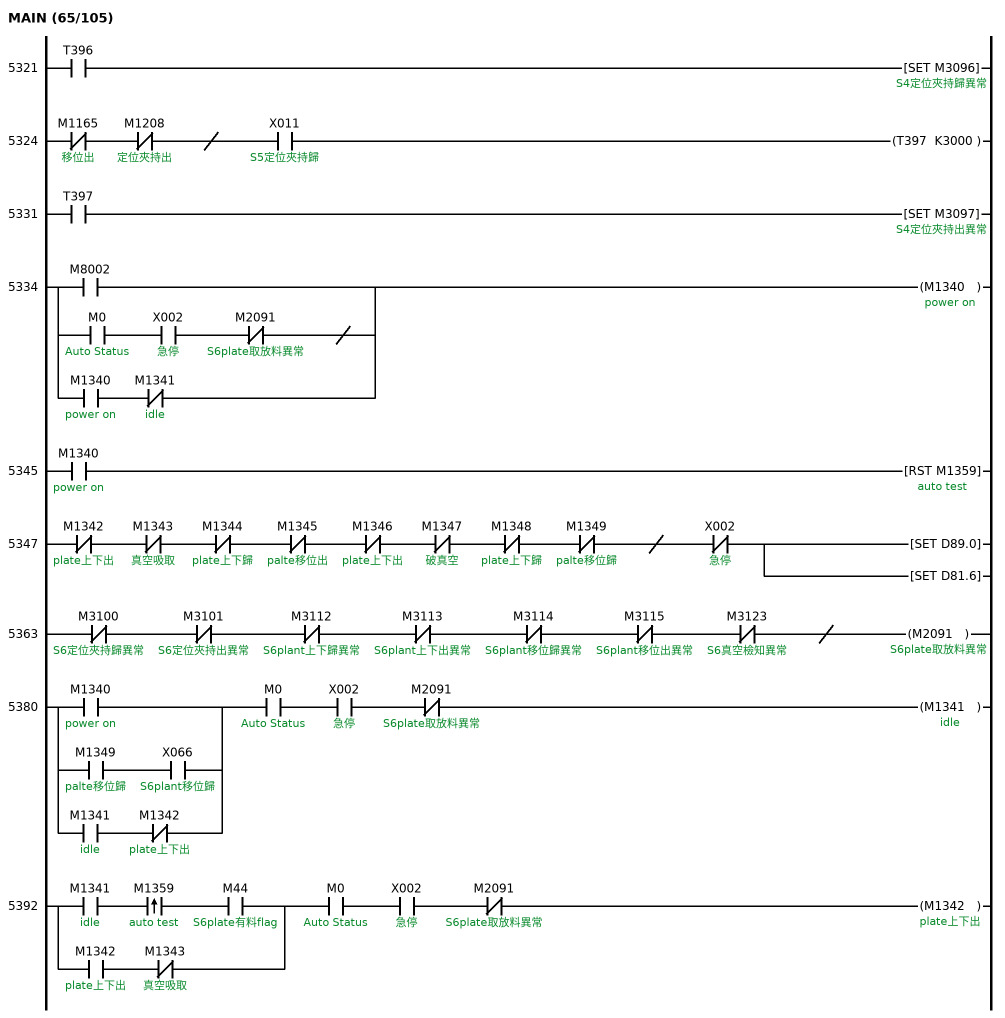
5321  LD      T396
      SET     M3096  ; S4定位夾持歸異常
5324  LDI     M1165  ; 移位出
      ANI     M1208  ; 定位夾持出
      INV
      AND     X011  ; S5定位夾持歸
      OUT     T397 K3000
5331  LD      T397
      SET     M3097  ; S4定位夾持出異常
5334  LD      M8002
      LD      M0  ; Auto Status
      AND     X002  ; 急停
      ANI     M2091  ; S6plate取放料異常
      INV
      ORB
      LD      M1340  ; power on
      ANI     M1341  ; idle
      ORB
      OUT     M1340  ; power on
5345  LD      M1340  ; power on
      RST     M1359  ; auto test
5347  LDI     M1342  ; plate上下出
      ANI     M1343  ; 真空吸取
      ANI     M1344  ; plate上下歸
      ANI     M1345  ; palte移位出
      ANI     M1346  ; plate上下出
      ANI     M1347  ; 破真空
      ANI     M1348  ; plate上下歸
      ANI     M1349  ; palte移位歸
      INV
      ANI     X002  ; 急停
      SET     D89.0
      SET     D81.6
5363  LDI     M3100  ; S6定位夾持歸異常
      ANI     M3101  ; S6定位夾持出異常
      ANI     M3112  ; S6plant上下歸異常
      ANI     M3113  ; S6plant上下出異常
      ANI     M3114  ; S6plant移位歸異常
      ANI     M3115  ; S6plant移位出異常
      ANI     M3123  ; S6真空檢知異常
      INV
      OUT     M2091  ; S6plate取放料異常
5380  LD      M1340  ; power on
      LD      M1349  ; palte移位歸
      AND     X066  ; S6plant移位歸
      ORB
      LD      M1341  ; idle
      ANI     M1342  ; plate上下出
      ORB
      AND     M0  ; Auto Status
      AND     X002  ; 急停
      ANI     M2091  ; S6plate取放料異常
      OUT     M1341  ; idle
5392  LD      M1341  ; idle
      ANDP    M1359  ; auto test
      AND     M44  ; S6plate有料flag
      LD      M1342  ; plate上下出
      ANI     M1343  ; 真空吸取
      ORB
      AND     M0  ; Auto Status
      AND     X002  ; 急停
      ANI     M2091  ; S6plate取放料異常
      OUT     M1342  ; plate上下出
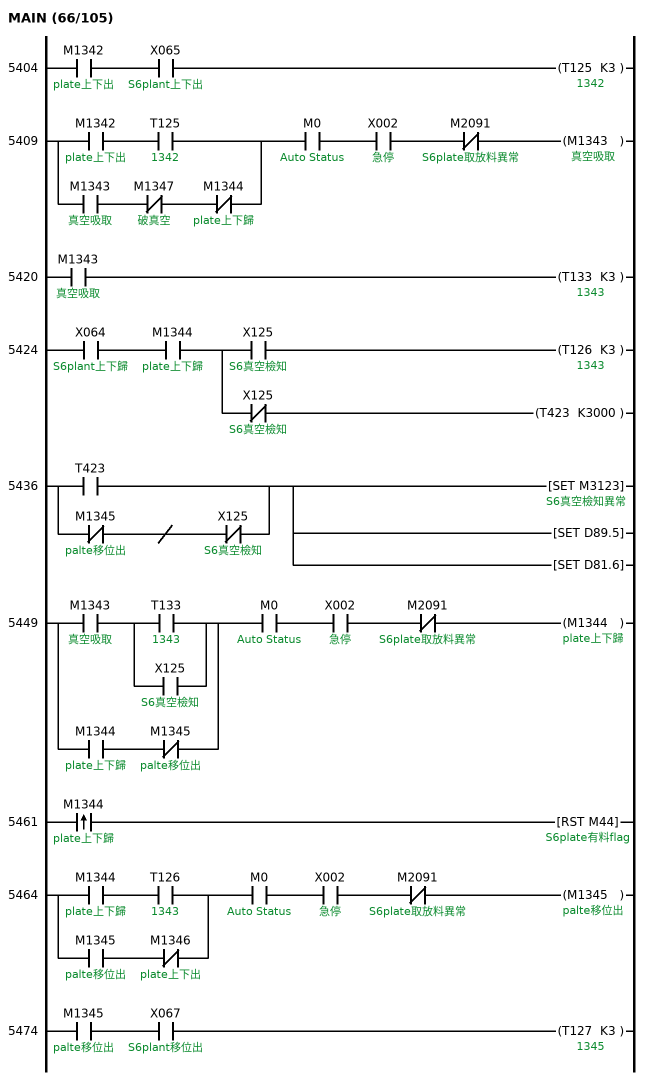
5404  LD      M1342  ; plate上下出
      AND     X065  ; S6plant上下出
      OUT     T125 K3  ; 1342
5409  LD      M1342  ; plate上下出
      AND     T125  ; 1342
      LD      M1343  ; 真空吸取
      ANI     M1347  ; 破真空
      ANI     M1344  ; plate上下歸
      ORB
      AND     M0  ; Auto Status
      AND     X002  ; 急停
      ANI     M2091  ; S6plate取放料異常
      OUT     M1343  ; 真空吸取
5420  LD      M1343  ; 真空吸取
      OUT     T133 K3  ; 1343
5424  LD      X064  ; S6plant上下歸
      AND     M1344  ; plate上下歸
      MPS
      AND     X125  ; S6真空檢知
      OUT     T126 K3  ; 1343
      MPP
      ANI     X125  ; S6真空檢知
      OUT     T423 K3000
5436  LD      T423
      LDI     M1345  ; palte移位出
      INV
      ANI     X125  ; S6真空檢知
      ORB
      SET     M3123  ; S6真空檢知異常
      SET     D89.5
      SET     D81.6
5449  LD      M1343  ; 真空吸取
      LD      T133  ; 1343
      OR      X125  ; S6真空檢知
      ANB
      LD      M1344  ; plate上下歸
      ANI     M1345  ; palte移位出
      ORB
      AND     M0  ; Auto Status
      AND     X002  ; 急停
      ANI     M2091  ; S6plate取放料異常
      OUT     M1344  ; plate上下歸
5461  LDP     M1344  ; plate上下歸
      RST     M44  ; S6plate有料flag
5464  LD      M1344  ; plate上下歸
      AND     T126  ; 1343
      LD      M1345  ; palte移位出
      ANI     M1346  ; plate上下出
      ORB
      AND     M0  ; Auto Status
      AND     X002  ; 急停
      ANI     M2091  ; S6plate取放料異常
      OUT     M1345  ; palte移位出
5474  LD      M1345  ; palte移位出
      AND     X067  ; S6plant移位出
      OUT     T127 K3  ; 1345
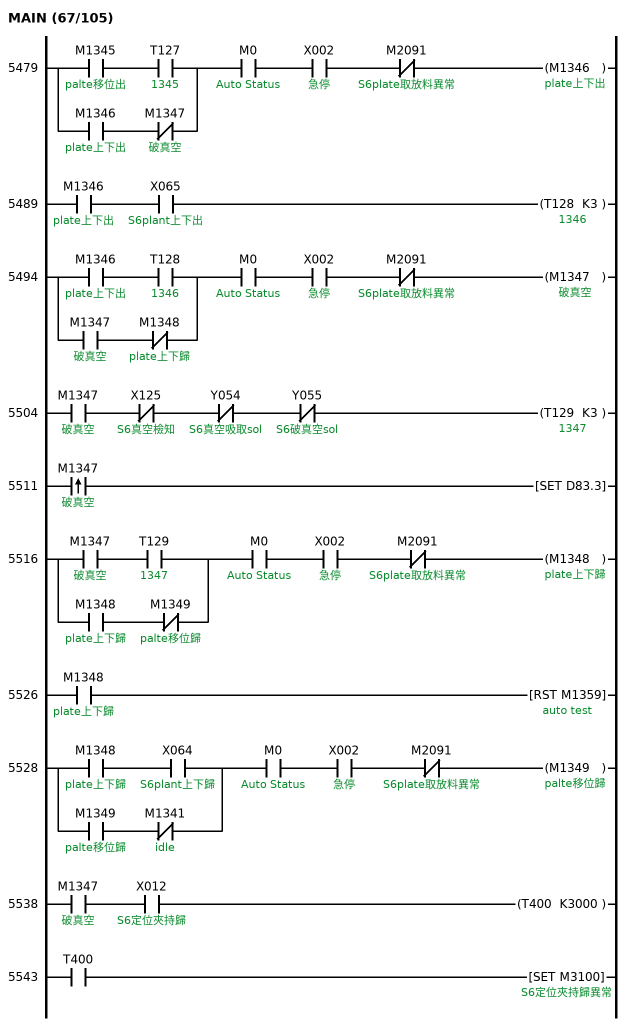
5479  LD      M1345  ; palte移位出
      AND     T127  ; 1345
      LD      M1346  ; plate上下出
      ANI     M1347  ; 破真空
      ORB
      AND     M0  ; Auto Status
      AND     X002  ; 急停
      ANI     M2091  ; S6plate取放料異常
      OUT     M1346  ; plate上下出
5489  LD      M1346  ; plate上下出
      AND     X065  ; S6plant上下出
      OUT     T128 K3  ; 1346
5494  LD      M1346  ; plate上下出
      AND     T128  ; 1346
      LD      M1347  ; 破真空
      ANI     M1348  ; plate上下歸
      ORB
      AND     M0  ; Auto Status
      AND     X002  ; 急停
      ANI     M2091  ; S6plate取放料異常
      OUT     M1347  ; 破真空
5504  LD      M1347  ; 破真空
      ANI     X125  ; S6真空檢知
      ANI     Y054  ; S6真空吸取sol
      ANI     Y055  ; S6破真空sol
      OUT     T129 K3  ; 1347
5511  LDP     M1347  ; 破真空
      SET     D83.3
5516  LD      M1347  ; 破真空
      AND     T129  ; 1347
      LD      M1348  ; plate上下歸
      ANI     M1349  ; palte移位歸
      ORB
      AND     M0  ; Auto Status
      AND     X002  ; 急停
      ANI     M2091  ; S6plate取放料異常
      OUT     M1348  ; plate上下歸
5526  LD      M1348  ; plate上下歸
      RST     M1359  ; auto test
5528  LD      M1348  ; plate上下歸
      AND     X064  ; S6plant上下歸
      LD      M1349  ; palte移位歸
      ANI     M1341  ; idle
      ORB
      AND     M0  ; Auto Status
      AND     X002  ; 急停
      ANI     M2091  ; S6plate取放料異常
      OUT     M1349  ; palte移位歸
5538  LD      M1347  ; 破真空
      AND     X012  ; S6定位夾持歸
      OUT     T400 K3000
5543  LD      T400
      SET     M3100  ; S6定位夾持歸異常
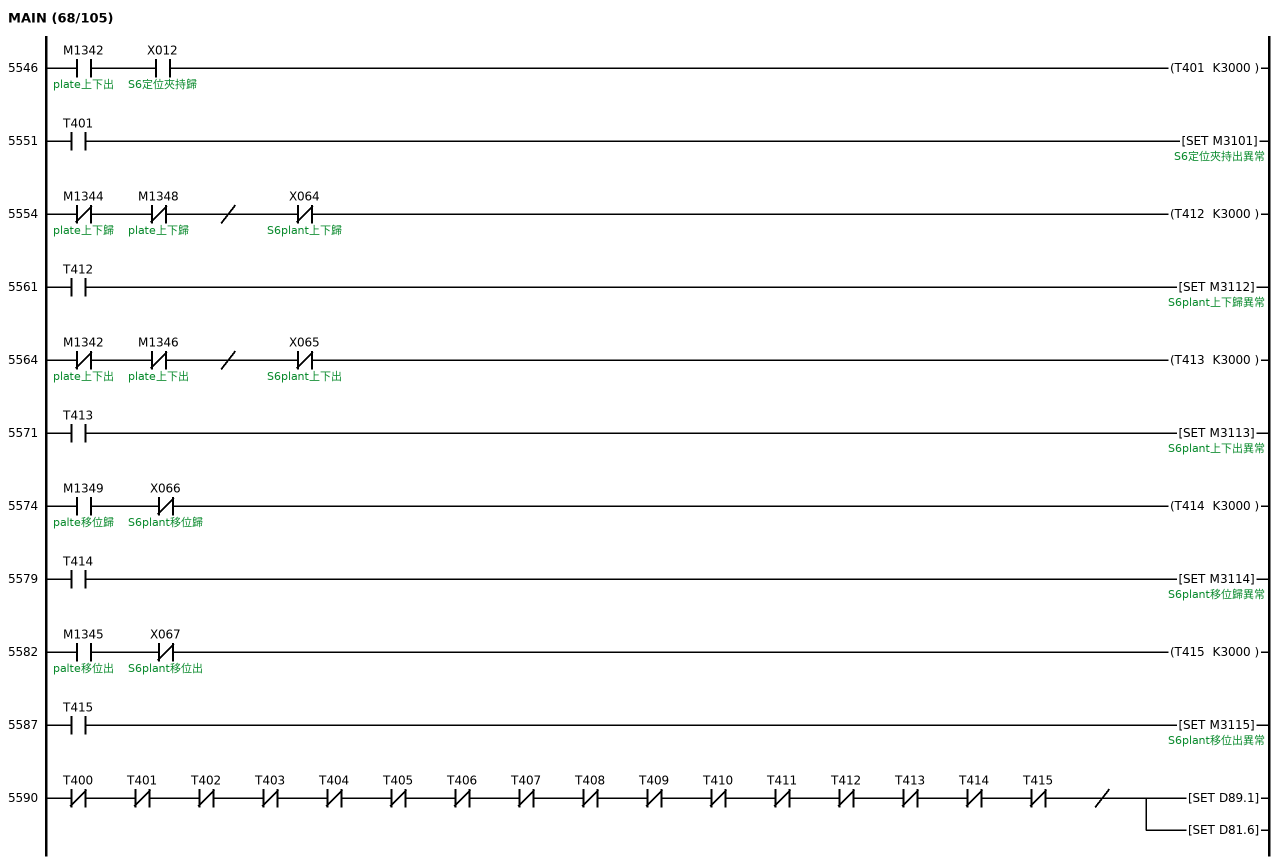
5546  LD      M1342  ; plate上下出
      AND     X012  ; S6定位夾持歸
      OUT     T401 K3000
5551  LD      T401
      SET     M3101  ; S6定位夾持出異常
5554  LDI     M1344  ; plate上下歸
      ANI     M1348  ; plate上下歸
      INV
      ANI     X064  ; S6plant上下歸
      OUT     T412 K3000
5561  LD      T412
      SET     M3112  ; S6plant上下歸異常
5564  LDI     M1342  ; plate上下出
      ANI     M1346  ; plate上下出
      INV
      ANI     X065  ; S6plant上下出
      OUT     T413 K3000
5571  LD      T413
      SET     M3113  ; S6plant上下出異常
5574  LD      M1349  ; palte移位歸
      ANI     X066  ; S6plant移位歸
      OUT     T414 K3000
5579  LD      T414
      SET     M3114  ; S6plant移位歸異常
5582  LD      M1345  ; palte移位出
      ANI     X067  ; S6plant移位出
      OUT     T415 K3000
5587  LD      T415
      SET     M3115  ; S6plant移位出異常
5590  LDI     T400
      ANI     T401
      ANI     T402
      ANI     T403
      ANI     T404
      ANI     T405
      ANI     T406
      ANI     T407
      ANI     T408
      ANI     T409
      ANI     T410
      ANI     T411
      ANI     T412
      ANI     T413
      ANI     T414
      ANI     T415
      INV
      SET     D89.1
      SET     D81.6
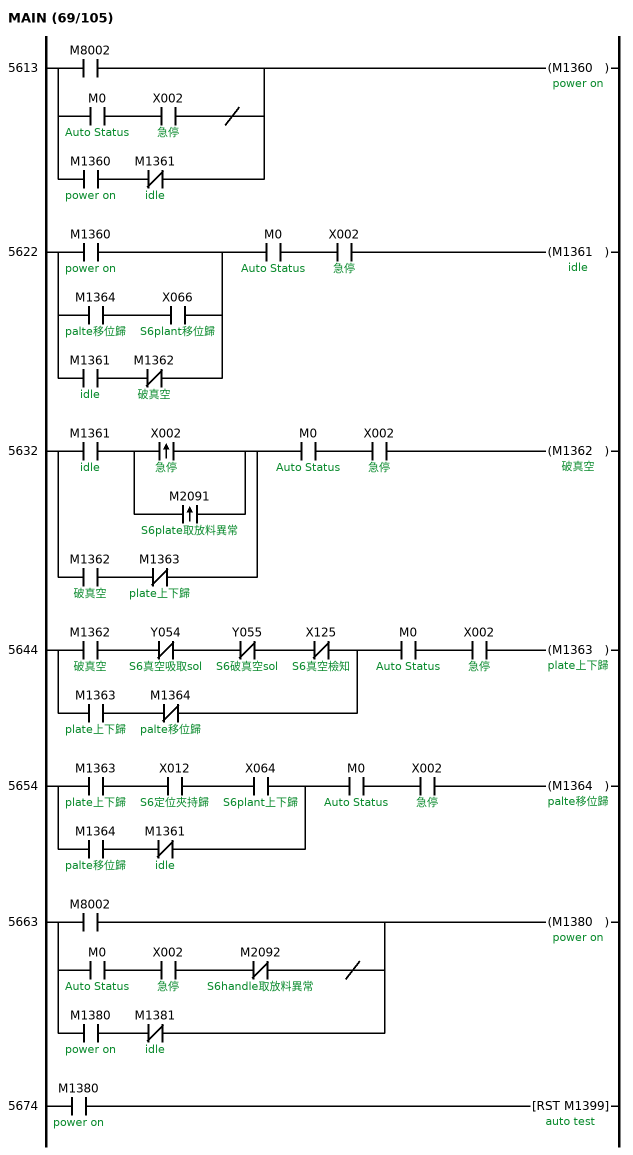
5613  LD      M8002
      LD      M0  ; Auto Status
      AND     X002  ; 急停
      INV
      ORB
      LD      M1360  ; power on
      ANI     M1361  ; idle
      ORB
      OUT     M1360  ; power on
5622  LD      M1360  ; power on
      LD      M1364  ; palte移位歸
      AND     X066  ; S6plant移位歸
      ORB
      LD      M1361  ; idle
      ANI     M1362  ; 破真空
      ORB
      AND     M0  ; Auto Status
      AND     X002  ; 急停
      OUT     M1361  ; idle
5632  LD      M1361  ; idle
      LDP     X002  ; 急停
      ORP     M2091  ; S6plate取放料異常
      ANB
      LD      M1362  ; 破真空
      ANI     M1363  ; plate上下歸
      ORB
      AND     M0  ; Auto Status
      AND     X002  ; 急停
      OUT     M1362  ; 破真空
5644  LD      M1362  ; 破真空
      ANI     Y054  ; S6真空吸取sol
      ANI     Y055  ; S6破真空sol
      ANI     X125  ; S6真空檢知
      LD      M1363  ; plate上下歸
      ANI     M1364  ; palte移位歸
      ORB
      AND     M0  ; Auto Status
      AND     X002  ; 急停
      OUT     M1363  ; plate上下歸
5654  LD      M1363  ; plate上下歸
      AND     X012  ; S6定位夾持歸
      AND     X064  ; S6plant上下歸
      LD      M1364  ; palte移位歸
      ANI     M1361  ; idle
      ORB
      AND     M0  ; Auto Status
      AND     X002  ; 急停
      OUT     M1364  ; palte移位歸
5663  LD      M8002
      LD      M0  ; Auto Status
      AND     X002  ; 急停
      ANI     M2092  ; S6handle取放料異常
      INV
      ORB
      LD      M1380  ; power on
      ANI     M1381  ; idle
      ORB
      OUT     M1380  ; power on
5674  LD      M1380  ; power on
      RST     M1399  ; auto test
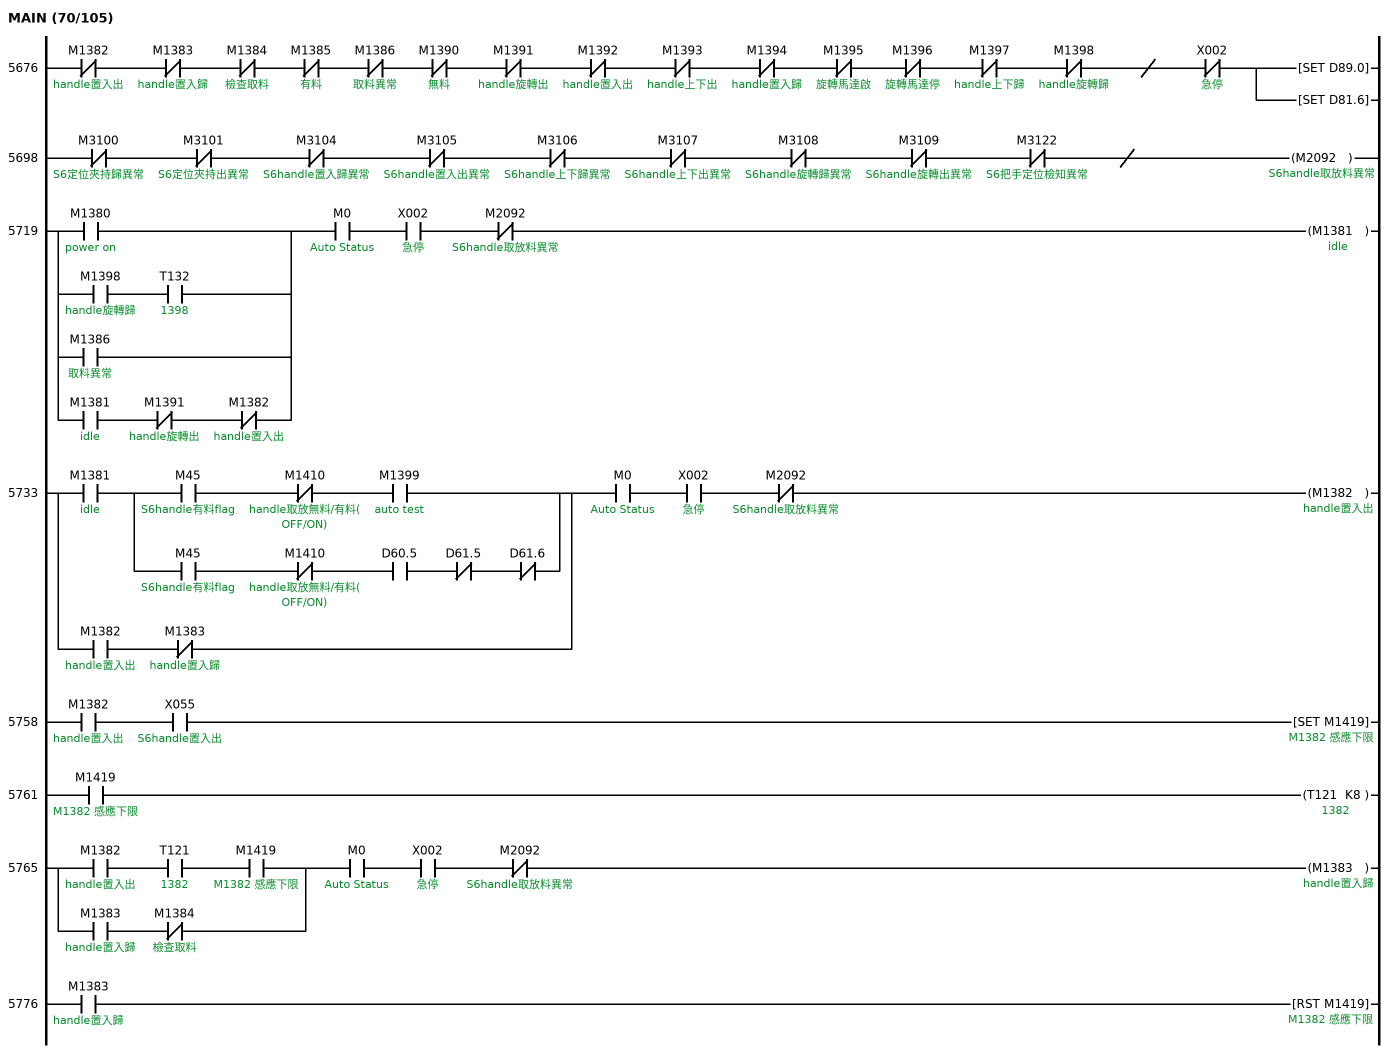
5676  LDI     M1382  ; handle置入出
      ANI     M1383  ; handle置入歸
      ANI     M1384  ; 檢查取料
      ANI     M1385  ; 有料
      ANI     M1386  ; 取料異常
      ANI     M1390  ; 無料
      ANI     M1391  ; handle旋轉出
      ANI     M1392  ; handle置入出
      ANI     M1393  ; handle上下出
      ANI     M1394  ; handle置入歸
      ANI     M1395  ; 旋轉馬達啟
      ANI     M1396  ; 旋轉馬達停
      ANI     M1397  ; handle上下歸
      ANI     M1398  ; handle旋轉歸
      INV
      ANI     X002  ; 急停
      SET     D89.0
      SET     D81.6
5698  LDI     M3100  ; S6定位夾持歸異常
      ANI     M3101  ; S6定位夾持出異常
      ANI     M3104  ; S6handle置入歸異常
      ANI     M3105  ; S6handle置入出異常
      ANI     M3106  ; S6handle上下歸異常
      ANI     M3107  ; S6handle上下出異常
      ANI     M3108  ; S6handle旋轉歸異常
      ANI     M3109  ; S6handle旋轉出異常
      ANI     M3122  ; S6把手定位檢知異常
      INV
      OUT     M2092  ; S6handle取放料異常
5719  LD      M1380  ; power on
      LD      M1398  ; handle旋轉歸
      AND     T132  ; 1398
      ORB
      OR      M1386  ; 取料異常
      LD      M1381  ; idle
      ANI     M1391  ; handle旋轉出
      ANI     M1382  ; handle置入出
      ORB
      AND     M0  ; Auto Status
      AND     X002  ; 急停
      ANI     M2092  ; S6handle取放料異常
      OUT     M1381  ; idle
5733  LD      M1381  ; idle
      LD      M45  ; S6handle有料flag
      ANI     M1410  ; handle取放無料/有料(OFF/ON)
      AND     M1399  ; auto test
      LD      M45  ; S6handle有料flag
      ANI     M1410  ; handle取放無料/有料(OFF/ON)
      AND     D60.5
      ANI     D61.5
      ANI     D61.6
      ORB
      ANB
      LD      M1382  ; handle置入出
      ANI     M1383  ; handle置入歸
      ORB
      AND     M0  ; Auto Status
      AND     X002  ; 急停
      ANI     M2092  ; S6handle取放料異常
      OUT     M1382  ; handle置入出
5758  LD      M1382  ; handle置入出
      AND     X055  ; S6handle置入出
      SET     M1419  ; M1382 感應下限
5761  LD      M1419  ; M1382 感應下限
      OUT     T121 K8  ; 1382
5765  LD      M1382  ; handle置入出
      AND     T121  ; 1382
      AND     M1419  ; M1382 感應下限
      LD      M1383  ; handle置入歸
      ANI     M1384  ; 檢查取料
      ORB
      AND     M0  ; Auto Status
      AND     X002  ; 急停
      ANI     M2092  ; S6handle取放料異常
      OUT     M1383  ; handle置入歸
5776  LD      M1383  ; handle置入歸
      RST     M1419  ; M1382 感應下限
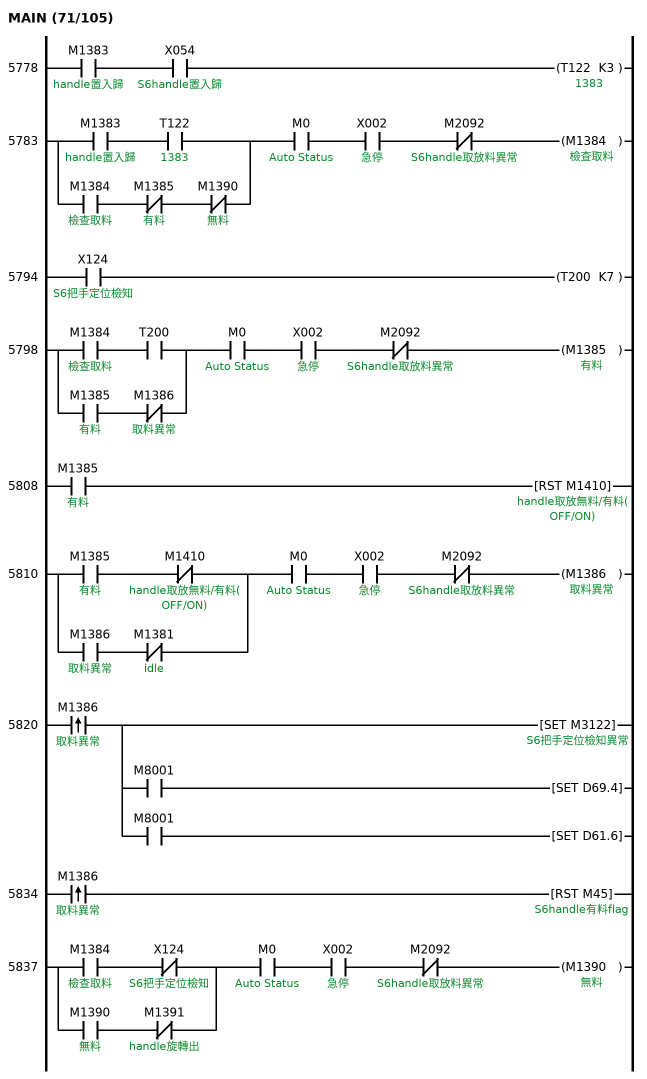
5778  LD      M1383  ; handle置入歸
      AND     X054  ; S6handle置入歸
      OUT     T122 K3  ; 1383
5783  LD      M1383  ; handle置入歸
      AND     T122  ; 1383
      LD      M1384  ; 檢查取料
      ANI     M1385  ; 有料
      ANI     M1390  ; 無料
      ORB
      AND     M0  ; Auto Status
      AND     X002  ; 急停
      ANI     M2092  ; S6handle取放料異常
      OUT     M1384  ; 檢查取料
5794  LD      X124  ; S6把手定位檢知
      OUT     T200 K7
5798  LD      M1384  ; 檢查取料
      AND     T200
      LD      M1385  ; 有料
      ANI     M1386  ; 取料異常
      ORB
      AND     M0  ; Auto Status
      AND     X002  ; 急停
      ANI     M2092  ; S6handle取放料異常
      OUT     M1385  ; 有料
5808  LD      M1385  ; 有料
      RST     M1410  ; handle取放無料/有料(OFF/ON)
5810  LD      M1385  ; 有料
      ANI     M1410  ; handle取放無料/有料(OFF/ON)
      LD      M1386  ; 取料異常
      ANI     M1381  ; idle
      ORB
      AND     M0  ; Auto Status
      AND     X002  ; 急停
      ANI     M2092  ; S6handle取放料異常
      OUT     M1386  ; 取料異常
5820  LDP     M1386  ; 取料異常
      SET     M3122  ; S6把手定位檢知異常
      MPS
      AND     M8001
      SET     D69.4
      MPP
      AND     M8001
      SET     D61.6
5834  LDP     M1386  ; 取料異常
      RST     M45  ; S6handle有料flag
5837  LD      M1384  ; 檢查取料
      ANI     X124  ; S6把手定位檢知
      LD      M1390  ; 無料
      ANI     M1391  ; handle旋轉出
      ORB
      AND     M0  ; Auto Status
      AND     X002  ; 急停
      ANI     M2092  ; S6handle取放料異常
      OUT     M1390  ; 無料
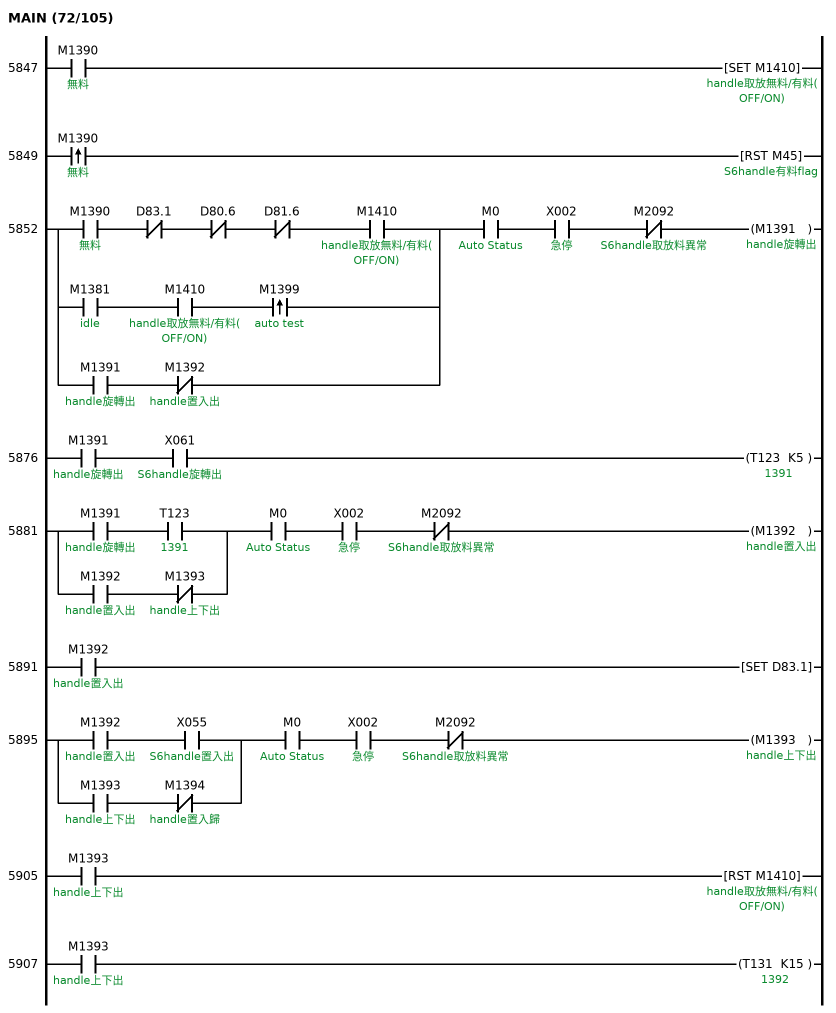
5847  LD      M1390  ; 無料
      SET     M1410  ; handle取放無料/有料(OFF/ON)
5849  LDP     M1390  ; 無料
      RST     M45  ; S6handle有料flag
5852  LD      M1390  ; 無料
      ANI     D83.1
      ANI     D80.6
      ANI     D81.6
      AND     M1410  ; handle取放無料/有料(OFF/ON)
      LD      M1381  ; idle
      AND     M1410  ; handle取放無料/有料(OFF/ON)
      ANDP    M1399  ; auto test
      ORB
      LD      M1391  ; handle旋轉出
      ANI     M1392  ; handle置入出
      ORB
      AND     M0  ; Auto Status
      AND     X002  ; 急停
      ANI     M2092  ; S6handle取放料異常
      OUT     M1391  ; handle旋轉出
5876  LD      M1391  ; handle旋轉出
      AND     X061  ; S6handle旋轉出
      OUT     T123 K5  ; 1391
5881  LD      M1391  ; handle旋轉出
      AND     T123  ; 1391
      LD      M1392  ; handle置入出
      ANI     M1393  ; handle上下出
      ORB
      AND     M0  ; Auto Status
      AND     X002  ; 急停
      ANI     M2092  ; S6handle取放料異常
      OUT     M1392  ; handle置入出
5891  LD      M1392  ; handle置入出
      SET     D83.1
5895  LD      M1392  ; handle置入出
      AND     X055  ; S6handle置入出
      LD      M1393  ; handle上下出
      ANI     M1394  ; handle置入歸
      ORB
      AND     M0  ; Auto Status
      AND     X002  ; 急停
      ANI     M2092  ; S6handle取放料異常
      OUT     M1393  ; handle上下出
5905  LD      M1393  ; handle上下出
      RST     M1410  ; handle取放無料/有料(OFF/ON)
5907  LD      M1393  ; handle上下出
      OUT     T131 K15  ; 1392
